# B&R Automation Studio project NewPendant_NG4_11_05_25A (part 3)

### Hardcoded.c
```c
/********************************************************************
 * COPYRIGHT -- wsi
 ********************************************************************
 * Package: Robot
 * File: Hardcoded.c
 * Author: wsi
 * Created: March 08, 2013
 *******************************************************************/
#ifndef _HARDCODED_C
#define _HARDCODED_C

#include <bur/plctypes.h>
#ifdef _DEFAULT_INCLUDES
	#include <AsDefault.h>
#endif

#include <..\GlobDef.h>
#include <..\GlobDecl.h>
#include <..\..\Lib\LCDLib.c>

//#include <string.h>

/**
char line[6][4] = {	{0xFF,0xFF,0xFF,0x00},
					{0xFF,0xFF,0xFF,0x00},
					{0xFF,0xFF,0xFF,0x00},
					{0xFF,0xFF,0xFF,0x00},
					{0xFF,0xFF,0xFF,0x00},
					{0xFF,0xFF,0xFF,0x00} };

char emptyLine[21] = { 0x20 , 0x00 };

**/

static	plcstring txt_example[32];
static	plcstring txt_hidden_example[32];

void HardCodeCFg(MASTER_typ *m);

void SetupNODES_Android(MASTER_typ *m , UDINT pNode ,UINT nodeNum );

void SetPageDict(PAGE_DICT_typ* dict , UINT indx , char* pTxt);

void SetupNODES_Android(MASTER_typ *m , UDINT pNode ,UINT nodeNum ){

int i, k , h , n;
char status;
Cfg_typ *cfg;
CurCfg_typ *curCfg;
CurCalib_typ *curCalib;
Scaled_Var_obj *var , *tempVar;

Enum_Var_obj  *enumVar;
Integer_Var_obj *intVar;

LCD_NODE_obj *node , *tempNode;
//LCD_MGR_obj *lcd;

	if(!m)
		return;

	if(!pNode)
		return;

	node = (LCD_NODE_obj*)pNode;
	cfg = (Cfg_typ*) m->pCfg;
	curCfg = (CurCfg_typ*) m->pCurCfg;
	var = (Scaled_Var_obj*) m->pScaledVar;
	curCalib = (CurCalib_typ*) m->pCalib;

	enumVar = cfg->EnumVar;

	if(!cfg || ! curCfg || !var || !curCalib)
		return;

	/************************************/

	n = 0;

	///// MENU ////////////
	/** P_MENU **/
	i = P_MENU;			h=varSTRING_HMI_0;
	SetPageDict(&cfg->PagesDict[n++] , P_MENU , "P_MENU");

	node[i].pHeadNode	= (UDINT)&node[P_MENU];
	node[i].Type = N_SCROLL   ;
	node[i].var.Type = T_STRING;
	node[i].var.Var1ID = varSTRING_curProgramName;
	strcpy(node[i++].var.Format, "Cur Program: %s");

	node[i].pHeadNode	= (UDINT)&node[P_MENU];
	node[i].Type = N_SCROLL;
	node[i].var.Type = T_STRING;
	node[i].var.Var1ID = varSTRING_NextProgramName;
	strcpy(node[i++].var.Format, "Next Program: %s");

	node[i].pHeadNode	= (UDINT)&node[P_MENU];
	node[i].Type = N_JUMP + N_EVENT;
	node[i].Event = EVNT_EDIT_PARAM_VAL;
	node[i].JumpLineID = 0;
	node[i].MinUserLevel = USER_OPERATOR;
	node[i].pJumpNode = (UDINT)&node[P_PARAM];
	strcpy(node[i++].var.Format, "Parameters Value");

	node[i].pHeadNode	= (UDINT)&node[P_MENU];
	node[i].Type = N_JUMP + N_EVENT;
	node[i].Event = EVNT_EDIT_PARAM_VAL;
	node[i].JumpLineID = 0;
	node[i].MinUserLevel = USER_OPERATOR;
	node[i].pJumpNode = (UDINT)&node[P_PARAM_BOOSTS];
	strcpy(node[i++].var.Format, "Parameters Boost");

	node[i].pHeadNode	= (UDINT)&node[P_MENU];
	node[i].Type = N_JUMP + N_EVENT;
	node[i].Event = EVNT_EDIT_PARAM_VAL;
	node[i].JumpLineID = 0;
	node[i].MinUserLevel = USER_OPERATOR;
	node[i].pJumpNode = (UDINT)&node[P_PARAM_CONTIN_WELD];
	strcpy(node[i++].var.Format, "Parameters Contin. Weld");

	node[i].pHeadNode	= (UDINT)&node[P_MENU];
	node[i].Type = N_JUMP;
	node[i].JumpLineID = 0;
	node[i].MinUserLevel = USER_OPERATOR;
	node[i].pJumpNode = (UDINT)&node[P_PAR_REVIEW];
	strcpy(node[i++].var.Format, "Timing Review");

	node[i].pHeadNode	= (UDINT)&node[P_MENU];
	node[i].Type = N_JUMP;
	node[i].JumpLineID = 0;
	node[i].MinUserLevel = USER_OPERATOR;
	node[i].pJumpNode = (UDINT)&node[P_VAR_SETUP];
	strcpy(node[i++].var.Format, "Var Unit Setup");

	node[i].pHeadNode	= (UDINT)&node[P_MENU];
	node[i].Type = N_JUMP;
	node[i].JumpLineID = 0;
	node[i].MinUserLevel = USER_OPERATOR;
	node[i].pJumpNode = (UDINT)&node[P_SPEC_OPERATION];
	strcpy(node[i++].var.Format, "Special Operation");

	node[i].pHeadNode 	= (UDINT)&node[P_MENU];
	node[i].Type = N_SCROLL + N_NO_PREFIX;
	node[i].var.Type = T_STRING;
	node[i].var.Var1ID = varSTRING_PlcVersion;
	strcpy(node[i++].var.Format, "%s");

	node[i].pHeadNode	= (UDINT)&node[P_MENU];
	node[i].Type = N_SCROLL + N_EVENT ;
	node[i].Event = EVNT_TOGGLE;
	node[i].var.Type = T_STRING;
	node[i].var.Var1ID = (h++);
	strcpy(node[i++].var.Format, "COOL PWR is: %s");

	node[i].pHeadNode	= (UDINT)&node[P_MENU];
	node[i].Type = N_SCROLL  + N_EDIT_IN_PLACE ;
	node[i].var.Type = T_STRING;
	node[i].var.Var1ID = (h++);
	strcpy(node[i++].var.Format, "COOL Sensor is: %s");

	node[i].pHeadNode	= (UDINT)&node[P_MENU];
	node[i].Type = N_SCROLL  + N_EDIT_IN_PLACE ;
	node[i].var.Type = T_STRING;
	node[i].var.Var1ID = (h++);
	strcpy(node[i++].var.Format, "GAS Sensor is: %s");

	////

	/*
	node[i].pHeadNode	= (UDINT)&node[P_MENU];
	node[i].Type = N_JUMP;
	node[i].JumpLineID = 0;
	node[i].MinUserLevel = USER_OPERATOR;
	node[i].pJumpNode = (UDINT)&node[P_SEGMENTS];
	strcpy(node[i++].var.Format, "Segments Setup");
	*/

	/** P_MODE_CALIB**/
	i = P_MODE_CALIB;			h=varSTRING_HMI_0;
	SetPageDict(&cfg->PagesDict[n++] , P_MODE_CALIB , "P_MODE_CALIB");

	node[i].pHeadNode	= (UDINT)&node[P_MODE_CALIB];
	node[i].Type = N_JUMP + N_EVENT;
	node[i].Event = EVNT_RETURN_CALIB_MODE;
	node[i].MinUserLevel = USER_OPERATOR;
	node[i].pJumpNode = (UDINT)&node[P_MENU];
	strcpy(node[i++].var.Format, "Return ");

	node[i].pHeadNode	= (UDINT)&node[P_MODE_CALIB];
	node[i].Type = N_JUMP + N_EVENT;
	node[i].Event = EVNT_GO_CALIB_MODE;
	node[i].JumpLineID = 0;
	node[i].pJumpNode = (UDINT)&node[P_MODE_TIG_PS_CALIB_PAR];
	strcpy(node[i++].var.Format, "TIG PS Calib.");

	node[i].pHeadNode	= (UDINT)&node[P_MODE_CALIB];
	node[i].Type = N_JUMP + N_EVENT;
	node[i].Event = EVNT_GO_CALIB_MODE;
	node[i].JumpLineID = 0;
	node[i].pJumpNode = (UDINT)&node[P_MODE_HW_PS_CALIB_PAR];
	strcpy(node[i++].var.Format, "HW PS Calib");

	node[i].pHeadNode	= (UDINT)&node[P_MODE_CALIB];
	node[i].Type = N_JUMP + N_EVENT;
	node[i].Event = EVNT_GO_CALIB_MODE;
	node[i].JumpLineID = 0;
	node[i].pJumpNode = (UDINT)&node[P_MODE_OSC_LIMIT_CALIB];
	strcpy(node[i++].var.Format, "OSC Limit Setup");

	node[i].pHeadNode	= (UDINT)&node[P_MODE_CALIB];
	node[i].Type = N_JUMP + N_EVENT;
	node[i].Event = EVNT_GO_CALIB_MODE;
	node[i].JumpLineID = 0;
	node[i].pJumpNode = (UDINT)&node[P_MODE_TIG_FBK_CALIB];
	strcpy(node[i++].var.Format, "ARC Volt FBK Calib");

	node[i].pHeadNode	= (UDINT)&node[P_MODE_CALIB];
	node[i].Type = N_JUMP + N_EVENT;
	node[i].Event = EVNT_GO_CALIB_MODE;
	node[i].JumpLineID = 0;
	node[i].pJumpNode = (UDINT)&node[P_MODE_TVL_CALIB_PAR];
	strcpy(node[i++].var.Format, "TVL Calib");

	node[i].pHeadNode	= (UDINT)&node[P_MODE_CALIB];
	node[i].Type = N_JUMP + N_EVENT;
	node[i].Event = EVNT_GO_CALIB_MODE;
	node[i].JumpLineID = 0;
	node[i].pJumpNode = (UDINT)&node[P_MODE_WF_CALIB_PAR];
	strcpy(node[i++].var.Format, "WFeed Calib");

	node[i].pHeadNode	= (UDINT)&node[P_MODE_CALIB];
	node[i].Type = N_JUMP + N_EVENT;
	node[i].Event = EVNT_VER_TIG_PS_CALIB;
	node[i].JumpLineID = 0;
	node[i].pJumpNode = (UDINT)&node[P_MODE_TIG_PS_CALIB_VER];
	strcpy(node[i++].var.Format, "TIG PS Test");

	node[i].pHeadNode	= (UDINT)&node[P_MODE_CALIB];
	node[i].Type = N_JUMP + N_EVENT;
	node[i].Event = EVNT_VER_HW_PS_CALIB;
	node[i].JumpLineID = 0;
	node[i].pJumpNode = (UDINT)&node[P_MODE_HW_PS_CALIB_VER];
	strcpy(node[i++].var.Format, "HW PS Test");

	node[i].pHeadNode	= (UDINT)&node[P_MODE_CALIB];
	node[i].Type = N_JUMP + N_EVENT;
	node[i].Event = EVNT_VER_TVL_CALIB;
	node[i].JumpLineID = 0;
	node[i].pJumpNode = (UDINT)&node[P_MODE_TVL_CALIB_VER];
	strcpy(node[i++].var.Format, "TVL Test");

	node[i].pHeadNode	= (UDINT)&node[P_MODE_CALIB];
	node[i].Type = N_JUMP + N_EVENT;
	node[i].Event = EVNT_VER_WF_CALIB;
	node[i].JumpLineID = 0;
	node[i].pJumpNode = (UDINT)&node[P_MODE_WF_CALIB_VER];
	strcpy(node[i++].var.Format, "WFeed Test");

	/** P_PARAM **/
	i = P_PARAM;			h=varSTRING_HMI_0;
	SetPageDict(&cfg->PagesDict[n++] , P_PARAM , "P_PARAM");

	node[i].pHeadNode	= (UDINT)&node[P_PARAM];
	node[i].Type = N_JUMP;
	node[i].JumpLineID = 0;
	node[i].pJumpNode = (UDINT)&node[P_MENU];
	strcpy(node[i++].var.Format, "Return ");

	node[i].pHeadNode	= (UDINT)&node[P_PARAM];
	node[i].Type = N_JUMP;
	node[i].JumpLineID = 0;
	node[i].pJumpNode = (UDINT)&node[P_PARAM_GAS];
	strcpy(node[i++].var.Format, "Param. GAS/COOL");

	node[i].pHeadNode	= (UDINT)&node[P_PARAM];
	node[i].Type = N_JUMP;
	node[i].JumpLineID = 0;
	node[i].pJumpNode = (UDINT)&node[P_PARAM_AVC];
	strcpy(node[i++].var.Format, "Param. AVC");

	node[i].pHeadNode	= (UDINT)&node[P_PARAM];
	node[i].Type = N_JUMP;
	node[i].JumpLineID = 0;
	node[i].pJumpNode = (UDINT)&node[P_PARAM_TIG];
	strcpy(node[i++].var.Format, "Param. TIG");

	node[i].pHeadNode	= (UDINT)&node[P_PARAM];
	node[i].Type = N_JUMP;
	node[i].JumpLineID = 0;
	node[i].pJumpNode = (UDINT)&node[P_PARAM_OSC];
	strcpy(node[i++].var.Format, "Param. OSC");

	node[i].pHeadNode	= (UDINT)&node[P_PARAM];
	node[i].Type = N_JUMP;
	node[i].JumpLineID = 0;
	node[i].pJumpNode = (UDINT)&node[P_PARAM_TVL_ROT];
	strcpy(node[i++].var.Format, "Param.TVL");

	node[i].pHeadNode	= (UDINT)&node[P_PARAM];
	node[i].Type = N_JUMP;
	node[i].JumpLineID = 0;
	node[i].pJumpNode = (UDINT)&node[P_PARAM_WF];
	strcpy(node[i++].var.Format, "Param. WF");

	node[i].pHeadNode	= (UDINT)&node[P_PARAM];
	node[i].Type = N_JUMP;
	node[i].JumpLineID = 0;
	node[i].pJumpNode = (UDINT)&node[P_PARAM_WP];
	strcpy(node[i++].var.Format, "Param. WP");

	node[i].pHeadNode	= (UDINT)&node[P_PARAM];
	node[i].Type = N_JUMP;
	node[i].JumpLineID = 0;
	node[i].pJumpNode = (UDINT)&node[P_PARAM_HW];
	strcpy(node[i++].var.Format, "Param. HW");

	node[i].pHeadNode	= (UDINT)&node[P_PARAM];
	node[i].Type = N_JUMP;
	node[i].JumpLineID = 0;
	node[i].pJumpNode = (UDINT)&node[P_PARAM_WRST];
	strcpy(node[i++].var.Format, "Param. WRIST");

	node[i].pHeadNode	= (UDINT)&node[P_PARAM];
	node[i].Type = N_JUMP;
	node[i].JumpLineID = 0;
	node[i].pJumpNode = (UDINT)&node[P_PARAM_INDX];
	strcpy(node[i++].var.Format, "Param. INDX");

	node[i].pHeadNode	= (UDINT)&node[P_PARAM];
	node[i].Type = N_EDIT;
	node[i].MinUserLevel = 5;
	node[i].var.Type = T_ENUM;
	node[i].var.Var1ID = parENUM_WeldProgramLinkMode;
	//strcpy(node[i++].var.Format, "Load Next Prg.: %s");
	strcpy(node[i++].var.Format, "%name%: %s");

	node[i].pHeadNode	= (UDINT)&node[P_PARAM];
	node[i].Type = N_EDIT;
	node[i].MinUserLevel = 5;
	node[i].var.Type = T_ENUM;
	node[i].var.Var1ID = parENUM_PathMode;
	//strcpy(node[i++].var.Format, "Swap Head: %s");
	strcpy(node[i++].var.Format, "%name%: %s");

	node[i].pHeadNode	= (UDINT)&node[P_PARAM];
	node[i].Type = N_EDIT;
	node[i].var.Type = T_SCALED;
	node[i].var.Var1ID = parGEN_WeldProgramRepeat;
	//strcpy(node[i++].var.Format, "Repeat: %s");
	strcpy(node[i++].var.Format, "%name%: %s");

	node[i].pHeadNode	= (UDINT)&node[P_PARAM];
	node[i].Type = N_SCROLL + N_EDIT_IN_PLACE;
	node[i].var.Type = T_STRING;
	node[i].var.Var1ID = (h++);
	strcpy(node[i++].var.Format, "%s");

	node[i].pHeadNode 	= (UDINT)&node[P_PARAM];
	node[i].Type = N_SCROLL + N_NO_PREFIX;
	node[i].MinUserLevel = 5;
	strcpy(node[i++].var.Format, "** SYNCH. options**");

	node[i].pHeadNode	= (UDINT)&node[P_PARAM];
	node[i].Type = N_EDIT;
	node[i].MinUserLevel = 5;
	node[i].var.Type = T_ENUM;
	node[i].var.Var1ID = parENUM_TIG_Mode;
	//strcpy(node[i++].var.Format, "TIG Mode: %s");
	strcpy(node[i++].var.Format, "%name%: %s");

	node[i].pHeadNode	= (UDINT)&node[P_PARAM];
	node[i].Type = N_EDIT;
	node[i].MinUserLevel = 5;
	node[i].var.Type = T_ENUM;
	node[i].var.Var1ID = parENUM_AVC_Mode;
	//strcpy(node[i++].var.Format, "AVC Mode: %s");
	strcpy(node[i++].var.Format, "%name%: %s");

	node[i].pHeadNode	= (UDINT)&node[P_PARAM];
	node[i].Type = N_EDIT;
	node[i].MinUserLevel = 5;
	node[i].var.Type = T_ENUM;
	node[i].var.Var1ID = parENUM_TVL_SYN_MODE;
	//strcpy(node[i++].var.Format, "TVL Synch. Mode: %s");
	strcpy(node[i++].var.Format, "%name%: %s");

	node[i].pHeadNode	= (UDINT)&node[P_PARAM];
	node[i].Type = N_EDIT;
	node[i].MinUserLevel = 5;
	node[i].var.Type = T_ENUM;
	node[i].var.Var1ID = parENUM_WF_SYN_MODE;
	//strcpy(node[i++].var.Format, "WF Synch. Mode: %s");
	strcpy(node[i++].var.Format, "%name%: %s");

	node[i].pHeadNode	= (UDINT)&node[P_PARAM];
	node[i].Type = N_EDIT;
	node[i].MinUserLevel = 5;
	node[i].var.Type = T_ENUM;
	node[i].var.Var1ID = parENUM_WP_SYN_MODE;
	//strcpy(node[i++].var.Format, "WP Synch. Mode: %s");
	strcpy(node[i++].var.Format, "%name%: %s");

	i = P_PARAM_APPL;			h=varSTRING_HMI_0;
	SetPageDict(&cfg->PagesDict[n++] , P_PARAM_APPL , "P_PARAM_APPL");

	node[i].pHeadNode	= (UDINT)&node[P_PARAM_APPL];
	node[i].Type = N_EDIT;
	node[i].MinUserLevel = 5;
	node[i].var.Type = T_SCALED;
	node[i].var.Var1ID = parTVL_RunDist;
	//strcpy(node[i++].var.Format, "RUN Dist: %s");
	strcpy(node[i++].var.Format, "%name%: %s");

	node[i].pHeadNode	= (UDINT)&node[P_PARAM_APPL];
	node[i].Type = N_SCROLL + N_EDIT_IN_PLACE;
	node[i].MinUserLevel = 5;
	node[i].var.Type = T_STRING;
	node[i].var.Var1ID = (h++);
	strcpy(node[i++].var.Format, "%s"); // Zone editor

	node[i].pHeadNode	= (UDINT)&node[P_PARAM_APPL];
	node[i].Type = N_SCROLL + N_EDIT_IN_PLACE;
	node[i].MinUserLevel = 5;
	node[i].var.Type = T_STRING;
	node[i].var.Var1ID = (h++);
	strcpy(node[i++].var.Format, "%s"); // Track Dia

	node[i].pHeadNode	= (UDINT)&node[P_PARAM_APPL];
	node[i].Type = N_EDIT;
	node[i].var.Type = T_SCALED;
	node[i].var.Var1ID = parTVL_TrackDia;
	//strcpy(node[i++].var.Format, "Tungsten Track Dia: %s");
	strcpy(node[i++].var.Format, "%name%: %s");

	node[i].pHeadNode	= (UDINT)&node[P_PARAM_APPL];
	node[i].Type = N_EDIT;
	node[i].MinUserLevel = 5;
	node[i].var.Type = T_ENUM;
	node[i].var.Var1ID = parENUM_WeldProgramLinkMode;
	//strcpy(node[i++].var.Format, "Load Next Prg.: %s");
	strcpy(node[i++].var.Format, "%name%: %s");

	node[i].pHeadNode	= (UDINT)&node[P_PARAM_APPL];
	node[i].Type = N_EDIT;
	node[i].MinUserLevel = 5;
	node[i].var.Type = T_ENUM;
	node[i].var.Var1ID = parENUM_PathMode;
	//strcpy(node[i++].var.Format, "Swap Head: %s");
	strcpy(node[i++].var.Format, "%name%: %s");

	node[i].pHeadNode	= (UDINT)&node[P_PARAM_APPL];
	node[i].Type = N_EDIT;
	node[i].var.Type = T_SCALED;
	node[i].var.Var1ID = parGEN_WeldProgramRepeat;
	//strcpy(node[i++].var.Format, "Repeat: %s");
	strcpy(node[i++].var.Format, "%name%: %s");

	node[i].pHeadNode	= (UDINT)&node[P_PARAM_APPL];
	node[i].Type = N_SCROLL + N_EDIT_IN_PLACE;
	node[i].MinUserLevel = 5;
	node[i].var.Type = T_STRING;
	node[i].var.Var1ID = (h++);
	strcpy(node[i++].var.Format, "%s"); // Weld Report ON / OFF

	node[i].pHeadNode	= (UDINT)&node[P_PARAM_APPL];
	node[i].Type = N_SCROLL + N_EDIT_IN_PLACE;
	node[i].MinUserLevel = 5;
	node[i].var.Type = T_STRING;
	node[i].var.Var1ID = (h++);
	strcpy(node[i++].var.Format, "%s"); // TVL Reverse RampDown ON / OFF

	/*
	node[i].pHeadNode	= (UDINT)&node[P_PARAM_APPL];
	node[i].Type = N_SCROLL + N_EVENT;
	node[i].Event = EVNT_OK;
	node[i].MinUserLevel = 5;
	node[i].var.Type = T_STRING;
	node[i].var.Var1ID = (h++);
	strcpy(node[i++].var.Format, "%s"); // Set Tilt Zero
	*/

	/** P_PARAM_WRST **/
	i = P_PARAM_WRST;			h=varSTRING_HMI_0;
	SetPageDict(&cfg->PagesDict[n++] , P_PARAM_WRST , "P_PARAM_WRST");

	node[i].pHeadNode	= (UDINT)&node[P_PARAM_WRST];
	node[i].Type = N_JUMP;
	node[i].JumpLineID = 0;
	node[i].pJumpNode = (UDINT)&node[P_PARAM];
	strcpy(node[i++].var.Format, "Return ");

	node[i].pHeadNode 	= (UDINT)&node[P_PARAM_WRST];
	node[i].Type = N_EDIT;
	node[i].MinUserLevel = 5;
	node[i].var.Type = T_SCALED;
	node[i].var.Var1ID = parWRST_JogSpeedDirCntrl;
	strcpy(node[i++].var.Format, "%name%: %s");

	node[i].pHeadNode 	= (UDINT)&node[P_PARAM_WRST];
	node[i].Type = N_EDIT;
	node[i].MinUserLevel = 5;
	node[i].var.Type = T_SCALED;
	node[i].var.Var1ID = parGEN_RadSpeed_Boost;
	strcpy(node[i++].var.Format, "%name%: %s");

	node[i].pHeadNode 	= (UDINT)&node[P_PARAM_WRST];
	node[i].Type = N_EDIT;
	node[i].MinUserLevel = 5;
	node[i].var.Type = T_SCALED;
	node[i].var.Var1ID = parTVL_POS_PREDICT;
	strcpy(node[i++].var.Format, "%name%: %s");

	node[i].pHeadNode	= (UDINT)&node[P_PARAM_WRST];
	node[i].Type = N_SCROLL;
	node[i].var.Type = T_STRING;
	node[i].var.Var1ID = (h++);
	strcpy(node[i++].var.Format, "%s");

	node[i].pHeadNode	= (UDINT)&node[P_PARAM_WRST];
	node[i].Type = N_SCROLL +  N_EVENT ;
	node[i].Event = EVNT_OK;
	node[i].var.Type = T_STRING;
	node[i].var.Var1ID = (h++);
	strcpy(node[i++].var.Format, "%s");

	/** P_PARAM_OSC **/
	i = P_PARAM_OSC;			h=varSTRING_HMI_0;
	SetPageDict(&cfg->PagesDict[n++] , P_PARAM_OSC , "P_PARAM_OSC");

	node[i].pHeadNode	= (UDINT)&node[P_PARAM_OSC];
	node[i].Type = N_JUMP;
	node[i].JumpLineID = 0;
	node[i].pJumpNode = (UDINT)&node[P_PARAM];
	strcpy(node[i++].var.Format, "Return ");

	node[i].pHeadNode 	= (UDINT)&node[P_PARAM_OSC];
	node[i].Type = N_EDIT;
	node[i].MinUserLevel = 5;
	node[i].var.Type = T_SCALED;
	node[i].var.Var1ID = parOSC_Amplit;
	//strcpy(node[i++].var.Format, "OSC WIDTH %s");
	strcpy(node[i++].var.Format, "%name%: %s");

	node[i].pHeadNode 	= (UDINT)&node[P_PARAM_OSC];
	node[i].Type = N_EDIT;
	node[i].MinUserLevel = 5;
	node[i].var.Type = T_SCALED;
	node[i].var.Var1ID = parOSC_Excur;
	//strcpy(node[i++].var.Format, "Excurs Tm.: %s");
	strcpy(node[i++].var.Format, "%name%: %s");

	node[i].pHeadNode 	= (UDINT)&node[P_PARAM_OSC];
	node[i].Type = N_EDIT;
	node[i].MinUserLevel = 5;
	node[i].var.Type = T_SCALED;
	node[i].var.Var1ID = parOSC_Dwell_In;
	//strcpy(node[i++].var.Format, "Dwell In: %s");
	strcpy(node[i++].var.Format, "%name%: %s");

	node[i].pHeadNode 	= (UDINT)&node[P_PARAM_OSC];
	node[i].Type = N_EDIT;
	node[i].MinUserLevel = 5;
	node[i].var.Type = T_SCALED;
	node[i].var.Var1ID = parOSC_Dwell_Out;
	//strcpy(node[i++].var.Format, "Dwell Out: %s");
	strcpy(node[i++].var.Format, "%name%: %s");

	node[i].pHeadNode 	= (UDINT)&node[P_PARAM_OSC];
	node[i].Type = N_SCROLL + N_NO_PREFIX;
	node[i].MinUserLevel = 5;
	strcpy(node[i++].var.Format, "******* MSC. *******");

	node[i].pHeadNode 	= (UDINT)&node[P_PARAM_OSC];
	node[i].Type = N_EDIT;
	node[i].MinUserLevel = 5;
	node[i].var.Type = T_SCALED;
	node[i].var.Var1ID = parOSC_InitAmplit;
	//strcpy(node[i++].var.Format, "OSC INI W %s");
	strcpy(node[i++].var.Format, "%name%: %s");

	node[i].pHeadNode 	= (UDINT)&node[P_PARAM_OSC];
	node[i].Type = N_EDIT;
	node[i].MinUserLevel = 5;
	node[i].var.Type = T_SCALED;
	node[i].var.Var1ID = parOSC_FinalAmplit;
	//strcpy(node[i++].var.Format, "OSC FIN W %s");
	strcpy(node[i++].var.Format, "%name%: %s");

	node[i].pHeadNode 	= (UDINT)&node[P_PARAM_OSC];
	node[i].Type = N_EDIT;
	node[i].MinUserLevel = 5;
	node[i].var.Type = T_ENUM;
	node[i].var.Var1ID = parENUM_OSC_Mode;
	strcpy(node[i++].var.Format, "%name%: %s");

	node[i].pHeadNode 	= (UDINT)&node[P_PARAM_OSC];
	node[i].Type = N_EDIT;
	node[i].MinUserLevel = 5;
	node[i].var.Type = T_ENUM;
	node[i].var.Var1ID = parENUM_OSC_Synch;
	strcpy(node[i++].var.Format, "%name%: %s");

	node[i].pHeadNode 	= (UDINT)&node[P_PARAM_OSC];
	node[i].Type = N_EDIT;
	node[i].MinUserLevel = 5;
	node[i].var.Type = T_SCALED;
	node[i].var.Var1ID = parOSC_Indx;
	strcpy(node[i++].var.Format, "%name%: %s");

	node[i].pHeadNode 	= (UDINT)&node[P_PARAM_OSC];
	node[i].Type = N_EDIT;
	node[i].MinUserLevel = 5;
	node[i].var.Type = T_SCALED;
	node[i].var.Var1ID = parOSC_Period;
	strcpy(node[i++].var.Format, "%name%: %s");

	node[i].pHeadNode 	= (UDINT)&node[P_PARAM_OSC];
	node[i].Type = N_EDIT;
	node[i].MinUserLevel = 5;
	node[i].var.Type = T_SCALED;
	node[i].var.Var1ID = parOSC_Indx_Vel;
	strcpy(node[i++].var.Format, "%name%: %s");

	node[i].pHeadNode 	= (UDINT)&node[P_PARAM_OSC];
	node[i].Type = N_EDIT;
	node[i].MinUserLevel = 5;
	node[i].var.Type = T_SCALED;
	node[i].var.Var1ID = parOSC_RampUpdate;
	//strcpy(node[i++].var.Format, "RampUpd.: %s");
	strcpy(node[i++].var.Format, "%name%: %s");

	node[i].pHeadNode	= (UDINT)&node[P_PARAM_OSC];
	node[i].Type = N_EDIT;
	node[i].MinUserLevel = 5;
	node[i].var.Type = T_SCALED;
	node[i].var.Var1ID = parOSC_JogSpeed;
	//strcpy(node[i++].var.Format, "Steer Speed: %s");
	strcpy(node[i++].var.Format, "%name%: %s");

	node[i].pHeadNode	= (UDINT)&node[P_PARAM_OSC];
	node[i].Type = N_EDIT;
	node[i].MinUserLevel = 5;
	node[i].var.Type = T_SCALED;
	node[i].var.Var1ID = parOSC_JogSpeedDirCntrl;
	//strcpy(node[i++].var.Format, "Jog Cntrl: %s");
	strcpy(node[i++].var.Format, "%name%: %s");

	node[i].pHeadNode 	= (UDINT)&node[P_PARAM_OSC];
	node[i].Type = N_EDIT;
	node[i].MinUserLevel = 5;
	node[i].var.Type = T_ENUM;
	node[i].var.Var1ID = parENUM_OSC_CAM;
	//strcpy(node[i++].var.Format, "Cam.: %s");
	strcpy(node[i++].var.Format, "%name%: %s");

	node[i].pHeadNode	= (UDINT)&node[P_PARAM_OSC];
	node[i].Type = N_EDIT;
	node[i].MinUserLevel = 5;
	node[i].var.Type = T_SCALED;
	node[i].var.Var1ID = parOSC_MaxTvlVel;
	//strcpy(node[i++].var.Format, "Max OSC Vel: %s");
	strcpy(node[i++].var.Format, "%name%: %s");

	node[i].pHeadNode 	= (UDINT)&node[P_PARAM_OSC];
	node[i].Type = N_SCROLL + N_NO_PREFIX;
	node[i].MinUserLevel = 5;
	strcpy(node[i++].var.Format, "**** CALCULATED ****");

	node[i].pHeadNode	= (UDINT)&node[P_PARAM_OSC];
	node[i].Type = N_EDIT;
	node[i].MinUserLevel = 5;
	node[i].var.Type = T_SCALED;
	node[i].var.Var1ID = parOSC_StartDly;
	//strcpy(node[i++].var.Format, "OSC DLY %s");
	strcpy(node[i++].var.Format, "%name%: %s");

	node[i].pHeadNode 	= (UDINT)&node[P_PARAM_OSC];
	node[i].Type = N_EDIT;
	node[i].MinUserLevel = 5;
	node[i].var.Type = T_SCALED;
	node[i].var.Var1ID = parOSC_RampUp;
	//strcpy(node[i++].var.Format, "O UPSCLOPE %s");
	strcpy(node[i++].var.Format, "%name%: %s");

	node[i].pHeadNode 	= (UDINT)&node[P_PARAM_OSC];
	node[i].Type = N_EDIT;
	node[i].MinUserLevel = 5;
	node[i].var.Type = T_SCALED;
	node[i].var.Var1ID = parOSC_StopDly;
	//strcpy(node[i++].var.Format, "O DS DLY %s");
	strcpy(node[i++].var.Format, "%name%: %s");

	node[i].pHeadNode 	= (UDINT)&node[P_PARAM_OSC];
	node[i].Type = N_EDIT;
	node[i].MinUserLevel = 5;
	node[i].var.Type = T_SCALED;
	node[i].var.Var1ID = parOSC_RampDwn;
	//strcpy(node[i++].var.Format, "O DWNSLOP %s");
	strcpy(node[i++].var.Format, "%name%: %s");

	/** P_PARAM_TVL_ROT **/
	i = P_PARAM_TVL_ROT;			h=varSTRING_HMI_0;
	SetPageDict(&cfg->PagesDict[n++] , P_PARAM_TVL_ROT , "P_PARAM_TVL_ROT");

	node[i].pHeadNode	= (UDINT)&node[P_PARAM_TVL_ROT];
	node[i].Type = N_JUMP;
	node[i].JumpLineID = 0;
	node[i].pJumpNode = (UDINT)&node[P_PARAM];
	strcpy(node[i++].var.Format, "Return ");

	node[i].pHeadNode 	= (UDINT)&node[P_PARAM_TVL_ROT];
	node[i].Type = N_EDIT;
	node[i].MinUserLevel = 5;
	node[i].var.Type = T_SCALED;
	node[i].var.Var1ID = parTVL_VelSP;
	node[i].var.Type = T_SCALED;
	//strcpy(node[i++].var.Format, "T PRI SP %s");
	strcpy(node[i++].var.Format, "%name%: %s");

	node[i].pHeadNode 	= (UDINT)&node[P_PARAM_TVL_ROT];
	node[i].Type = N_EDIT;
	node[i].MinUserLevel = 5;
	node[i].var.Type = T_SCALED;
	node[i].var.Var1ID = parTVL_VelInSP;
	node[i].var.Type = T_SCALED;
	//strcpy(node[i++].var.Format, "T PRI IN SP %s");
	strcpy(node[i++].var.Format, "%name%: %s");

	node[i].pHeadNode 	= (UDINT)&node[P_PARAM_TVL_ROT];
	node[i].Type = N_EDIT;
	node[i].MinUserLevel = 5;
	node[i].var.Type = T_SCALED;
	node[i].var.Var1ID = parTVL_VelOutSP;
	node[i].var.Type = T_SCALED;
	//strcpy(node[i++].var.Format, "T PRI OUT SP %s");
	strcpy(node[i++].var.Format, "%name%: %s");

	node[i].pHeadNode 	= (UDINT)&node[P_PARAM_TVL_ROT];
	node[i].Type = N_EDIT;
	node[i].MinUserLevel = 5;
	node[i].var.Type = T_SCALED;
	node[i].var.Var1ID = parTVL_VelBackSP;
	node[i].var.Type = T_SCALED;
	//strcpy(node[i++].var.Format, "T BCKG SP %s");
	strcpy(node[i++].var.Format, "%name%: %s");

	node[i].pHeadNode	= (UDINT)&node[P_PARAM_TVL_ROT];
	node[i].Type = N_EDIT;
	node[i].MinUserLevel = 5;
	node[i].var.Type = T_SCALED;
	node[i].var.Var1ID = parTVL_OverlapDist;
	//strcpy(node[i++].var.Format, "OVERLAP DIST: %s");
	strcpy(node[i++].var.Format, "%name%: %s");

	node[i].pHeadNode 	= (UDINT)&node[P_PARAM_TVL_ROT];
	node[i].Type = N_SCROLL + N_NO_PREFIX;
	node[i].MinUserLevel = 5;
	strcpy(node[i++].var.Format, "******* MSC. *******");

	node[i].pHeadNode 	= (UDINT)&node[P_PARAM_TVL_ROT];
	node[i].Type = N_EDIT;
	node[i].MinUserLevel = 5;
	node[i].var.Type = T_SCALED;
	node[i].var.Var1ID = parTVL_InitVel;
	node[i].var.Type = T_SCALED;
	//strcpy(node[i++].var.Format, "T INI SP %s");
	strcpy(node[i++].var.Format, "%name%: %s");

	node[i].pHeadNode 	= (UDINT)&node[P_PARAM_TVL_ROT];
	node[i].Type = N_EDIT;
	node[i].MinUserLevel = 5;
	node[i].var.Type = T_SCALED;
	node[i].var.Var1ID = parTVL_FinalVel;
	node[i].var.Type = T_SCALED;
	//strcpy(node[i++].var.Format, "T FIN SP %s");
	strcpy(node[i++].var.Format, "%name%: %s");

	node[i].pHeadNode 	= (UDINT)&node[P_PARAM_TVL_ROT];
	node[i].Type = N_EDIT;
	node[i].MinUserLevel = 5;
	node[i].var.Type = T_SCALED;
	node[i].var.Var1ID = parTVL_RampUpdate;
	//strcpy(node[i++].var.Format, "RampUpd.: %s");
	strcpy(node[i++].var.Format, "%name%: %s");

	node[i].pHeadNode	= (UDINT)&node[P_PARAM_TVL_ROT];
	node[i].Type = N_EDIT;
	node[i].MinUserLevel = 5;
	node[i].var.Type = T_SCALED;
	node[i].var.Var1ID = parTVL_JogSpeedDirCntrl;
	//strcpy(node[i++].var.Format, "Jog Cntrl: %s");
	strcpy(node[i++].var.Format, "%name%: %s");

	node[i].pHeadNode	= (UDINT)&node[P_PARAM_TVL_ROT];
	node[i].Type = N_EDIT;
	node[i].MinUserLevel = 5;
	node[i].var.Type = T_SCALED;
	node[i].var.Var1ID = parTVL_RewrapVel;
	//strcpy(node[i++].var.Format, "REWRP SP %s");
	strcpy(node[i++].var.Format, "%name%: %s");

	node[i].pHeadNode	= (UDINT)&node[P_PARAM_TVL_ROT];
	node[i].Type = N_EDIT;
	node[i].MinUserLevel = 5;
	node[i].var.Type = T_ENUM;
	node[i].var.Var1ID = parENUM_TVL_MODE;
	//strcpy(node[i++].var.Format, "TVL Mode: %s");
	strcpy(node[i++].var.Format, "%name%: %s");

	node[i].pHeadNode	= (UDINT)&node[P_PARAM_TVL_ROT];
	node[i].Type = N_EDIT;
	node[i].MinUserLevel = 5;
	node[i].var.Type = T_SCALED;
	node[i].var.Var1ID = parTVL_Jog2Stop;
	//strcpy(node[i++].var.Format, "Jog2Stop: %s");
	strcpy(node[i++].var.Format, "%name%: %s");

	node[i].pHeadNode	= (UDINT)&node[P_PARAM_TVL_ROT];
	node[i].Type = N_EDIT;
	node[i].MinUserLevel = 5;
	node[i].var.Type = T_SCALED;
	node[i].var.Var1ID = parTVL_SpeedTolerane;
	//strcpy(node[i++].var.Format, "Vel Toler: %s");
	strcpy(node[i++].var.Format, "%name%: %s");

	node[i].pHeadNode	= (UDINT)&node[P_PARAM_TVL_ROT];
	node[i].Type = N_EDIT;
	node[i].var.Type = T_SCALED;
	node[i].var.Var1ID = parTVL_CalibVel1;
	//strcpy(node[i++].var.Format, "Cal Vel1: %s");
	strcpy(node[i++].var.Format, "%name%: %s");

	node[i].pHeadNode	= (UDINT)&node[P_PARAM_TVL_ROT];
	node[i].Type = N_EDIT;
	node[i].var.Type = T_SCALED;
	node[i].var.Var1ID = parTVL_CalibVel2;
	//strcpy(node[i++].var.Format, "Cal Vel2: %s");
	strcpy(node[i++].var.Format, "%name%: %s");

	node[i].pHeadNode	= (UDINT)&node[P_PARAM_TVL_ROT];
	node[i].Type = N_EDIT;
	node[i].var.Type = T_SCALED;
	node[i].var.Var1ID = parTVL_TrackDia;
	//strcpy(node[i++].var.Format, "Tungsten Track Dia: %s");
	strcpy(node[i++].var.Format, "%name%: %s");

	node[i].pHeadNode	= (UDINT)&node[P_PARAM_TVL_ROT];
	node[i].Type = N_SCROLL + N_NO_PREFIX;
	node[i].MinUserLevel = 5;
	strcpy(node[i++].var.Format, "**** CALCULATED ****");

	node[i].pHeadNode 	= (UDINT)&node[P_PARAM_TVL_ROT];
	node[i].Type = N_EDIT;
	node[i].MinUserLevel = 5;
	node[i].var.Type = T_SCALED;
	node[i].var.Var1ID = parTVL_StartDly;
	//strcpy(node[i++].var.Format, "TVL DLY %s");
	strcpy(node[i++].var.Format, "%name%: %s");

	node[i].pHeadNode 	= (UDINT)&node[P_PARAM_TVL_ROT];
	node[i].Type = N_EDIT;
	node[i].MinUserLevel = 5;
	node[i].var.Type = T_SCALED;
	node[i].var.Var1ID = parTVL_RampUp;
	//strcpy(node[i++].var.Format, "T_UPSLOPE %s");
	strcpy(node[i++].var.Format, "%name%: %s");

	node[i].pHeadNode 	= (UDINT)&node[P_PARAM_TVL_ROT];
	node[i].Type = N_EDIT;
	node[i].MinUserLevel = 5;
	node[i].var.Type = T_SCALED;
	node[i].var.Var1ID = parTVL_StopDly;
	//strcpy(node[i++].var.Format, "T DS DLY %s");
	strcpy(node[i++].var.Format, "%name%: %s");

	node[i].pHeadNode 	= (UDINT)&node[P_PARAM_TVL_ROT];
	node[i].Type = N_EDIT;
	node[i].MinUserLevel = 5;
	node[i].var.Type = T_SCALED;
	node[i].var.Var1ID = parTVL_RampDwn;
	//strcpy(node[i++].var.Format, "T DWNSLOP %s");
	strcpy(node[i++].var.Format, "%name%: %s");

	node[i].pHeadNode	= (UDINT)&node[P_PARAM_TVL_ROT];
	node[i].Type = N_EDIT;
	node[i].MinUserLevel = 5;
	node[i].var.Type = T_SCALED;
	node[i].var.Var1ID = parTVL_RewrapDly;
	//strcpy(node[i++].var.Format, "REWRP DLY %s");
	strcpy(node[i++].var.Format, "%name%: %s");

	node[i].pHeadNode	= (UDINT)&node[P_PARAM_TVL_ROT];
	node[i].Type = N_EDIT;
	node[i].MinUserLevel = 5;
	node[i].var.Type = T_SCALED;
	node[i].var.Var1ID = parTVL_RunDist;
	//strcpy(node[i++].var.Format, "RUN Dist: %s");
	strcpy(node[i++].var.Format, "%name%: %s");

	node[i].pHeadNode	= (UDINT)&node[P_PARAM_TVL_ROT];
	node[i].Type = N_EDIT;
	node[i].MinUserLevel = 5;
	node[i].var.Type = T_SCALED;
	node[i].var.Var1ID = parTVL_BalanceDist;
	//strcpy(node[i++].var.Format, "Balance Dist: %s");
	strcpy(node[i++].var.Format, "%name%: %s");

	node[i].pHeadNode	= (UDINT)&node[P_PARAM_TVL_ROT];
	node[i].Type = N_EDIT;
	node[i].MinUserLevel = 5;
	node[i].var.Type = T_SCALED;
	node[i].var.Var1ID = parTVL_ZigZagDist;
	//strcpy(node[i++].var.Format, "ZigZag Dist: %s");
	strcpy(node[i++].var.Format, "%name%: %s");

	/** P_PARAM_WP **/
	i = P_PARAM_WP;			h=varSTRING_HMI_0;
	SetPageDict(&cfg->PagesDict[n++] , P_PARAM_WP , "P_PARAM_WP");

	node[i].pHeadNode	= (UDINT)&node[P_PARAM_WP];
	node[i].Type = N_JUMP;
	node[i].JumpLineID = 0;
	node[i].pJumpNode = (UDINT)&node[P_PARAM];
	strcpy(node[i++].var.Format, "Return ");

	node[i].pHeadNode	= (UDINT)&node[P_PARAM_WP];
	node[i].Type = N_EDIT;
	node[i].MinUserLevel = 5;
	node[i].var.Type = T_SCALED;
	node[i].var.Var1ID = parWP_SpeedSP;
	//strcpy(node[i++].var.Format, "WP FRG SP %s");
	strcpy(node[i++].var.Format, "%name% %s");

	node[i].pHeadNode	= (UDINT)&node[P_PARAM_WP];
	node[i].Type = N_EDIT;
	node[i].MinUserLevel = 5;
	node[i].var.Type = T_SCALED;
	node[i].var.Var1ID = parWP_SpeedInSP;
	//strcpy(node[i++].var.Format, "WP FRG IN SP %s");
	strcpy(node[i++].var.Format, "%name% %s");

	node[i].pHeadNode	= (UDINT)&node[P_PARAM_WP];
	node[i].Type = N_EDIT;
	node[i].MinUserLevel = 5;
	node[i].var.Type = T_SCALED;
	node[i].var.Var1ID = parWP_SpeedOutSP;
	//strcpy(node[i++].var.Format, "WP FRG OUT SP %s");
	strcpy(node[i++].var.Format, "%name%: %s");

	node[i].pHeadNode	= (UDINT)&node[P_PARAM_WP];
	node[i].Type = N_EDIT;
	node[i].MinUserLevel = 5;
	node[i].var.Type = T_SCALED;
	node[i].var.Var1ID = parWP_BkgSpeedSP;
	//strcpy(node[i++].var.Format, "WP BKG SP %s");
	strcpy(node[i++].var.Format, "%name%: %s");

	node[i].pHeadNode 	= (UDINT)&node[P_PARAM_WP];
	node[i].Type = N_SCROLL;
	node[i].MinUserLevel = 5;
	strcpy(node[i++].var.Format, "******* MSC. *******");

	node[i].pHeadNode	= (UDINT)&node[P_PARAM_WP];
	node[i].Type = N_EDIT;
	node[i].MinUserLevel = 5;
	node[i].var.Type = T_SCALED;
	node[i].var.Var1ID = parWP_SpeedInit;
	//strcpy(node[i++].var.Format, "WP INI SP %s");
	strcpy(node[i++].var.Format, "%name% %s");

	node[i].pHeadNode	= (UDINT)&node[P_PARAM_WP];
	node[i].Type = N_EDIT;
	node[i].MinUserLevel = 5;
	node[i].var.Type = T_SCALED;
	node[i].var.Var1ID = parWP_SpeedFinal;
	//strcpy(node[i++].var.Format, "WP FIN SP %s");
	strcpy(node[i++].var.Format, "%name%: %s");

	node[i].pHeadNode	= (UDINT)&node[P_PARAM_WP];
	node[i].Type = N_EDIT;
	node[i].MinUserLevel = 5;
	node[i].var.Type = T_SCALED;
	node[i].var.Var1ID = parWP_RampUpdate;
	//strcpy(node[i++].var.Format, "RampUpdate: %s");
	strcpy(node[i++].var.Format, "%name%: %s");

	/*
	node[i].pHeadNode	= (UDINT)&node[P_PARAM_WP];
	node[i].Type = N_EDIT;
	node[i].MinUserLevel = 5;
	node[i].var.Type = T_SCALED;
	node[i].var.Var1ID = parWP_Boost1SP;
	//strcpy(node[i++].var.Format, "Boost1: %s");
	strcpy(node[i++].var.Format, "%name% %s");

	node[i].pHeadNode	= (UDINT)&node[P_PARAM_WP];
	node[i].Type = N_EDIT;
	node[i].MinUserLevel = 5;
	node[i].var.Type = T_SCALED;
	node[i].var.Var1ID = parWP_Boost2SP;
	//strcpy(node[i++].var.Format, "Boost2: %s");
	strcpy(node[i++].var.Format, "%name% %s");
	*/

	node[i].pHeadNode	= (UDINT)&node[P_PARAM_WP];
	node[i].Type = N_EDIT;
	node[i].MinUserLevel = 5;
	node[i].var.Type = T_SCALED;
	node[i].var.Var1ID = parWP_JogSpeed;
	//strcpy(node[i++].var.Format, "Jog Vel.: %s");
	strcpy(node[i++].var.Format, "%name%: %s");

	node[i].pHeadNode	= (UDINT)&node[P_PARAM_WP];
	node[i].Type = N_EDIT;
	node[i].MinUserLevel = 5;
	node[i].var.Type = T_SCALED;
	node[i].var.Var1ID = parWP_JogSpeedDirCntrl;
	//strcpy(node[i++].var.Format, "Jog Cntrl: %s");
	strcpy(node[i++].var.Format, "%name%: %s");

	node[i].pHeadNode	= (UDINT)&node[P_PARAM_WP];
	node[i].Type = N_EDIT;
	node[i].MinUserLevel = 5;
	node[i].var.Type = T_ENUM;
	node[i].var.Var1ID = parENUM_WF_WP_Relation;
	//strcpy(node[i++].var.Format, "WP Auto Calc.: %s");
	strcpy(node[i++].var.Format, "%name% %s");

	node[i].pHeadNode	= (UDINT)&node[P_PARAM_WP];
	node[i].Type = N_SCROLL + N_NO_PREFIX;
	node[i].MinUserLevel = 5;
	strcpy(node[i++].var.Format, "**** CALCULATED ****");

	node[i].pHeadNode	= (UDINT)&node[P_PARAM_WP];
	node[i].Type = N_EDIT;
	node[i].MinUserLevel = 5;
	node[i].var.Type = T_SCALED;
	node[i].var.Var1ID = parWP_StartDly;
	//strcpy(node[i++].var.Format, "WP DLY %s");
	strcpy(node[i++].var.Format, "%name%: %s");

	node[i].pHeadNode	= (UDINT)&node[P_PARAM_WP];
	node[i].Type = N_EDIT;
	node[i].MinUserLevel = 5;
	node[i].var.Type = T_SCALED;
	node[i].var.Var1ID = parWP_RampUp;
	//strcpy(node[i++].var.Format, "WP UPSLOP %s");
	strcpy(node[i++].var.Format, "%name%: %s");

	node[i].pHeadNode	= (UDINT)&node[P_PARAM_WP];
	node[i].Type = N_EDIT;
	node[i].MinUserLevel = 5;
	node[i].var.Type = T_SCALED;
	node[i].var.Var1ID = parWP_StopDly;
	//strcpy(node[i++].var.Format, "WP DS DLY %s");
	strcpy(node[i++].var.Format, "%name%: %s");

	node[i].pHeadNode	= (UDINT)&node[P_PARAM_WP];
	node[i].Type = N_EDIT;
	node[i].MinUserLevel = 5;
	node[i].var.Type = T_SCALED;
	node[i].var.Var1ID = parWP_RampDwn;
	//strcpy(node[i++].var.Format, "WP DWNSLP %s");
	strcpy(node[i++].var.Format, "%name%: %s");

	/** P_PARAM_WF **/
	i = P_PARAM_WF;			h=varSTRING_HMI_0;
	SetPageDict(&cfg->PagesDict[n++] , P_PARAM_WF , "P_PARAM_WF");

	node[i].pHeadNode	= (UDINT)&node[P_PARAM_WF];
	node[i].Type = N_JUMP;
	node[i].JumpLineID = 0;
	node[i].pJumpNode = (UDINT)&node[P_PARAM];
	strcpy(node[i++].var.Format, "Return ");

	node[i].pHeadNode	= (UDINT)&node[P_PARAM_WF];
	node[i].Type = N_EDIT;
	node[i].MinUserLevel = 5;
	node[i].var.Type = T_SCALED;
	node[i].var.Var1ID = parWF_SpeedSP;
	//strcpy(node[i++].var.Format, "WF FRG SP %s");
	strcpy(node[i++].var.Format, "%name%: %s");

	node[i].pHeadNode	= (UDINT)&node[P_PARAM_WF];
	node[i].Type = N_EDIT;
	node[i].MinUserLevel = 5;
	node[i].var.Type = T_SCALED;
	node[i].var.Var1ID = parWF_SpeedInSP;
	//strcpy(node[i++].var.Format, "WF FRG IN SP %s");
	strcpy(node[i++].var.Format, "%name%: %s");

	node[i].pHeadNode	= (UDINT)&node[P_PARAM_WF];
	node[i].Type = N_EDIT;
	node[i].MinUserLevel = 5;
	node[i].var.Type = T_SCALED;
	node[i].var.Var1ID = parWF_SpeedOutSP;
	//strcpy(node[i++].var.Format, "WF FRG OUT SP %s");
	strcpy(node[i++].var.Format, "%name%: %s");

	node[i].pHeadNode	= (UDINT)&node[P_PARAM_WF];
	node[i].Type = N_EDIT;
	node[i].MinUserLevel = 5;
	node[i].var.Type = T_SCALED;
	node[i].var.Var1ID = parWF_BkgSpeedSP;
	//strcpy(node[i++].var.Format, "WF BKG SP %s");
	strcpy(node[i++].var.Format, "%name%: %s");

	node[i].pHeadNode 	= (UDINT)&node[P_PARAM_WF];
	node[i].Type = N_SCROLL + N_NO_PREFIX;
	node[i].MinUserLevel = 5;
	strcpy(node[i++].var.Format, "******* MSC. *******");

	node[i].pHeadNode	= (UDINT)&node[P_PARAM_WF];
	node[i].Type = N_EDIT;
	node[i].MinUserLevel = 5;
	node[i].var.Type = T_SCALED;
	node[i].var.Var1ID = parWF_SpeedInit;
	//strcpy(node[i++].var.Format, "WF INI SP %s");
	strcpy(node[i++].var.Format, "%name%: %s");

	node[i].pHeadNode	= (UDINT)&node[P_PARAM_WF];
	node[i].Type = N_EDIT;
	node[i].MinUserLevel = 5;
	node[i].var.Type = T_SCALED;
	node[i].var.Var1ID = parWF_SpeedFinal;
	//strcpy(node[i++].var.Format, "WF FIN SP %s");
	strcpy(node[i++].var.Format, "%name%: %s");

	node[i].pHeadNode	= (UDINT)&node[P_PARAM_WF];
	node[i].Type = N_EDIT;
	node[i].MinUserLevel = 5;
	node[i].var.Type = T_SCALED;
	node[i].var.Var1ID = parWF_RetractSpeed;
	//strcpy(node[i++].var.Format, "WF RET SP %s");
	strcpy(node[i++].var.Format, "%name%: %s");

	node[i].pHeadNode	= (UDINT)&node[P_PARAM_WF];
	node[i].Type = N_EDIT;
	node[i].MinUserLevel = 5;
	node[i].var.Type = T_SCALED;
	node[i].var.Var1ID = parWF_RetracDist;
	//strcpy(node[i++].var.Format, "WF UP LEN %s");
	strcpy(node[i++].var.Format, "%name%: %s");

	node[i].pHeadNode	= (UDINT)&node[P_PARAM_WF];
	node[i].Type = N_EDIT;
	node[i].MinUserLevel = 5;
	node[i].var.Type = T_SCALED;
	node[i].var.Var1ID = parWF_RampUpdate;
	//strcpy(node[i++].var.Format, "RampUpdate: %s");
	strcpy(node[i++].var.Format, "%name%: %s");

	node[i].pHeadNode	= (UDINT)&node[P_PARAM_WF];
	node[i].Type = N_EDIT;
	node[i].MinUserLevel = 5;
	node[i].var.Type = T_ENUM;
	node[i].var.Var1ID = parENUM_WF_AUX;
	strcpy(node[i++].var.Format, "%name%: %s");

	/*
	node[i].pHeadNode	= (UDINT)&node[P_PARAM_WF];
	node[i].Type = N_EDIT;
	node[i].MinUserLevel = 5;
	node[i].var.Type = T_SCALED;
	node[i].var.Var1ID = parWF_Boost1SP;
	//strcpy(node[i++].var.Format, "Boost1: %s");
	strcpy(node[i++].var.Format, "%name%: %s");

	node[i].pHeadNode	= (UDINT)&node[P_PARAM_WF];
	node[i].Type = N_EDIT;
	node[i].MinUserLevel = 5;
	node[i].var.Type = T_SCALED;
	node[i].var.Var1ID = parWF_Boost2SP;
	//strcpy(node[i++].var.Format, "Boost2: %s");
	strcpy(node[i++].var.Format, "%name%: %s");
	*/

	node[i].pHeadNode	= (UDINT)&node[P_PARAM_WF];
	node[i].Type = N_EDIT;
	node[i].MinUserLevel = 5;
	node[i].var.Type = T_SCALED;
	node[i].var.Var1ID = parWF_JogSpeed;
	//strcpy(node[i++].var.Format, "Jog Vel.: %s");
	strcpy(node[i++].var.Format, "%name%: %s");

	node[i].pHeadNode	= (UDINT)&node[P_PARAM_WF];
	node[i].Type = N_EDIT;
	node[i].MinUserLevel = 5;
	node[i].var.Type = T_SCALED;
	node[i].var.Var1ID = parWF_JogSpeedDirCntrl;
	//strcpy(node[i++].var.Format, "Jog Cntrl: %s");
	strcpy(node[i++].var.Format, "%name%: %s");

	node[i].pHeadNode	= (UDINT)&node[P_PARAM_WF];
	node[i].Type = N_EDIT;
	node[i].MinUserLevel = 5;
	node[i].var.Type = T_SCALED;
	node[i].var.Var1ID = parWF_CalibVel1;
	//strcpy(node[i++].var.Format, "Cal.Vel1: %s");
	strcpy(node[i++].var.Format, "%name%: %s");

	node[i].pHeadNode	= (UDINT)&node[P_PARAM_WF];
	node[i].Type = N_EDIT;
	node[i].MinUserLevel = 5;
	node[i].var.Type = T_SCALED;
	node[i].var.Var1ID = parWF_CalibVel2;
	//strcpy(node[i++].var.Format, "Cal.Vel2: %s");
	strcpy(node[i++].var.Format, "%name%: %s");

	node[i].pHeadNode	= (UDINT)&node[P_PARAM_WF];
	node[i].Type = N_SCROLL + N_NO_PREFIX;
	node[i].MinUserLevel = 5;
	strcpy(node[i++].var.Format, "**** CALCULATED ****");

	node[i].pHeadNode	= (UDINT)&node[P_PARAM_WF];
	node[i].Type = N_EDIT;
	node[i].MinUserLevel = 5;
	node[i].var.Type = T_SCALED;
	node[i].var.Var1ID = parWF_StartDly;
	//strcpy(node[i++].var.Format, "WF DLY %s");
	strcpy(node[i++].var.Format, "%name%: %s");

	node[i].pHeadNode	= (UDINT)&node[P_PARAM_WF];
	node[i].Type = N_EDIT;
	node[i].MinUserLevel = 5;
	node[i].var.Type = T_SCALED;
	node[i].var.Var1ID = parWF_RampUp;
	//strcpy(node[i++].var.Format, "WF UPSLOP %s");
	strcpy(node[i++].var.Format, "%name%: %s");

	node[i].pHeadNode	= (UDINT)&node[P_PARAM_WF];
	node[i].Type = N_EDIT;
	node[i].MinUserLevel = 5;
	node[i].var.Type = T_SCALED;
	node[i].var.Var1ID = parWF_StopDly;
	//strcpy(node[i++].var.Format, "WF DS DLY %s");
	strcpy(node[i++].var.Format, "%name%: %s");

	node[i].pHeadNode	= (UDINT)&node[P_PARAM_WF];
	node[i].Type = N_EDIT;
	node[i].MinUserLevel = 5;
	node[i].var.Type = T_SCALED;
	node[i].var.Var1ID = parWF_RampDwn;
	//strcpy(node[i++].var.Format, "WF DWNSLP %s");
	strcpy(node[i++].var.Format, "%name%: %s");

	node[i].pHeadNode	= (UDINT)&node[P_PARAM_WF];
	node[i].Type = N_EDIT;
	node[i].MinUserLevel = 5;
	node[i].var.Type = T_SCALED;
	node[i].var.Var1ID = parWF_RetractDly;
	//strcpy(node[i++].var.Format, "WFRET DLY %s");
	strcpy(node[i++].var.Format, "%name%: %s");

	/** P_PARAM_AVC **/
	i = P_PARAM_AVC;			h=varSTRING_HMI_0;
	SetPageDict(&cfg->PagesDict[n++] , P_PARAM_AVC , "P_PARAM_AVC");

	node[i].pHeadNode	= (UDINT)&node[P_PARAM_AVC];
	node[i].Type = N_JUMP;
	node[i].JumpLineID = 0;
	node[i].pJumpNode = (UDINT)&node[P_PARAM];
	strcpy(node[i++].var.Format, "Return ");

	node[i].pHeadNode	= (UDINT)&node[P_PARAM_AVC];
	node[i].Type = N_EDIT;
	node[i].MinUserLevel = 5;
	node[i].var.Type = T_SCALED;
	node[i].var.Var1ID = parAVC_VoltSP;
	//strcpy(node[i++].var.Format, "PRI VOLTS %s");
	strcpy(node[i++].var.Format, "%name%: %s");

	node[i].pHeadNode	= (UDINT)&node[P_PARAM_AVC];
	node[i].Type = N_EDIT;
	node[i].MinUserLevel = 5;
	node[i].var.Type = T_SCALED;
	node[i].var.Var1ID = parAVC_VoltInSP;
	//strcpy(node[i++].var.Format, "PRI IN VOLTS %s");
	strcpy(node[i++].var.Format, "%name%: %s");

	node[i].pHeadNode	= (UDINT)&node[P_PARAM_AVC];
	node[i].Type = N_EDIT;
	node[i].MinUserLevel = 5;
	node[i].var.Type = T_SCALED;
	node[i].var.Var1ID = parAVC_VoltOutSP;
	//strcpy(node[i++].var.Format, "PRI OUT VOLTS %s");
	strcpy(node[i++].var.Format, "%name%: %s");

	node[i].pHeadNode	= (UDINT)&node[P_PARAM_AVC];
	node[i].Type = N_EDIT;
	node[i].MinUserLevel = 5;
	node[i].var.Type = T_SCALED;
	node[i].var.Var1ID = parAVC_VoltBackSP;
	//strcpy(node[i++].var.Format, "BACK VOLTS %s");
	strcpy(node[i++].var.Format, "%name%: %s");

	node[i].pHeadNode	= (UDINT)&node[P_PARAM_AVC];
	node[i].Type = N_EDIT;
	node[i].MinUserLevel = 5;
	node[i].var.Type = T_ENUM;
	node[i].var.Var1ID = parENUM_AVC_Mode;
	//strcpy(node[i++].var.Format, "Mode: %s");
	strcpy(node[i++].var.Format, "%name%: %s");

	node[i].pHeadNode 	= (UDINT)&node[P_PARAM_AVC];
	node[i].Type = N_SCROLL + N_NO_PREFIX;
	node[i].MinUserLevel = 5;
	strcpy(node[i++].var.Format, "** ARC Start/Stop **");

	node[i].pHeadNode	= (UDINT)&node[P_PARAM_AVC];
	node[i].Type = N_EDIT;
	node[i].MinUserLevel = 5;
	node[i].var.Type = T_SCALED;
	node[i].var.Var1ID = parAVC_TouchVolt;
	//strcpy(node[i++].var.Format, "TOUCH V %s");
	strcpy(node[i++].var.Format, "%name%: %s");

	node[i].pHeadNode	= (UDINT)&node[P_PARAM_AVC];
	node[i].Type = N_EDIT;
	node[i].MinUserLevel = 5;
	node[i].var.Type = T_SCALED;
	node[i].var.Var1ID = parAVC_VoltInit;
	//strcpy(node[i++].var.Format, "AVC INI V %s");
	strcpy(node[i++].var.Format, "%name%: %s");

	node[i].pHeadNode	= (UDINT)&node[P_PARAM_AVC];
	node[i].Type = N_EDIT;
	node[i].MinUserLevel = 5;
	node[i].var.Type = T_SCALED;
	node[i].var.Var1ID = parAVC_TouchVel;
	//strcpy(node[i++].var.Format, "AVC SRI %s");
	strcpy(node[i++].var.Format, "%name%: %s");

	node[i].pHeadNode	= (UDINT)&node[P_PARAM_AVC];
	node[i].Type = N_EDIT;
	node[i].MinUserLevel = 5;
	node[i].var.Type = T_SCALED;
	node[i].var.Var1ID = parAVC_KissTm;
	//strcpy(node[i++].var.Format, "Touch Time %s");
	strcpy(node[i++].var.Format, "%name%: %s");

	node[i].pHeadNode	= (UDINT)&node[P_PARAM_AVC];
	node[i].Type = N_EDIT;
	node[i].MinUserLevel = 5;
	node[i].var.Type = T_SCALED;
	node[i].var.Var1ID = parAVC_ToSPVel;
	//strcpy(node[i++].var.Format, "AVC LU SP %s");
	strcpy(node[i++].var.Format, "%name%: %s");

	node[i].pHeadNode	= (UDINT)&node[P_PARAM_AVC];
	node[i].Type = N_EDIT;
	node[i].MinUserLevel = 5;
	node[i].var.Type = T_SCALED;
	node[i].var.Var1ID = parAVC_LU_TM;
	//strcpy(node[i++].var.Format, "AVC LU TM %s");
	strcpy(node[i++].var.Format, "%name%: %s");

	node[i].pHeadNode	= (UDINT)&node[P_PARAM_AVC];
	node[i].Type = N_EDIT;
	node[i].MinUserLevel = 5;
	node[i].var.Type = T_SCALED;
	node[i].var.Var1ID = parAVC_VoltFinal;
	//strcpy(node[i++].var.Format, "FIN VOLTS %s");
	strcpy(node[i++].var.Format, "%name%: %s");

	node[i].pHeadNode	= (UDINT)&node[P_PARAM_AVC];
	node[i].Type = N_EDIT;
	node[i].MinUserLevel = 5;
	node[i].var.Type = T_SCALED;
	node[i].var.Var1ID = parAVC_GoBackTm;
	//strcpy(node[i++].var.Format, "AVC UP TM %s");
	strcpy(node[i++].var.Format, "%name%: %s");

	node[i].pHeadNode	= (UDINT)&node[P_PARAM_AVC];
	node[i].Type = N_EDIT;
	node[i].MinUserLevel = 5;
	node[i].var.Type = T_SCALED;
	node[i].var.Var1ID = parAVC_LiftSpeedDirCntrl;
	//strcpy(node[i++].var.Format, "AVC UP SP %s");
	strcpy(node[i++].var.Format, "%name%: %s");

	node[i].pHeadNode	= (UDINT)&node[P_PARAM_AVC];
	node[i].Type = N_EDIT;
	node[i].MinUserLevel = 5;
	node[i].var.Type = T_SCALED;
	node[i].var.Var1ID = parAVC_TouchTm;
	//strcpy(node[i++].var.Format, "Touch TMO: %s");
	strcpy(node[i++].var.Format, "%name%: %s");

	node[i].pHeadNode	= (UDINT)&node[P_PARAM_AVC];
	node[i].Type = N_EDIT;
	node[i].MinUserLevel = 5;
	node[i].var.Type = T_SCALED;
	node[i].var.Var1ID = parAVC_TRetractTm;
	//strcpy(node[i++].var.Format, "Retract: %s");
	strcpy(node[i++].var.Format, "%name%: %s");

	node[i].pHeadNode	= (UDINT)&node[P_PARAM_AVC];
	node[i].Type = N_EDIT;
	node[i].MinUserLevel = 5;
	node[i].var.Type = T_SCALED;
	node[i].var.Var1ID = parAVC_TouchRepeat;
	//strcpy(node[i++].var.Format, "Repeat Cnt: %s");
	strcpy(node[i++].var.Format, "%name%: %s");

	/*
	node[i].pHeadNode 	= (UDINT)&node[P_PARAM_AVC];
	node[i].Type = N_SCROLL + N_NO_PREFIX;
	node[i].MinUserLevel = 5;
	strcpy(node[i++].var.Format, "******* MSC. *******");
	*/

	node[i].pHeadNode	= (UDINT)&node[P_PARAM_AVC];
	node[i].Type = N_EDIT;
	node[i].MinUserLevel = 5;
	node[i].var.Type = T_SCALED;
	node[i].var.Var1ID = parAVC_StartDly;
	//strcpy(node[i++].var.Format, "V UPS DLY %s");
	strcpy(node[i++].var.Format, "%name%: %s");

	node[i].pHeadNode	= (UDINT)&node[P_PARAM_AVC];
	node[i].Type = N_EDIT;
	node[i].MinUserLevel = 5;
	node[i].var.Type = T_SCALED;
	node[i].var.Var1ID = parAVC_VSPTmOut;
	//strcpy(node[i++].var.Format, "Init Volt Tmo: %s");
	strcpy(node[i++].var.Format, "%name%: %s");

	node[i].pHeadNode	= (UDINT)&node[P_PARAM_AVC];
	node[i].Type = N_EDIT;
	node[i].MinUserLevel = 5;
	node[i].var.Type = T_SCALED;
	node[i].var.Var1ID = parAVC_MaxVoltError;
	//strcpy(node[i++].var.Format, "Max Volt Err: %s");
	strcpy(node[i++].var.Format, "%name%: %s");

	node[i].pHeadNode	= (UDINT)&node[P_PARAM_AVC];
	node[i].Type = N_EDIT;
	node[i].MinUserLevel = 5;
	node[i].var.Type = T_SCALED;
	node[i].var.Var1ID = parAVC_JogSpeedDirCntrl;
	//strcpy(node[i++].var.Format, "Jog Cntrl: %s");
	strcpy(node[i++].var.Format, "%name%: %s");

	/*
	node[i].pHeadNode	= (UDINT)&node[P_PARAM_AVC];
	node[i].Type = N_EDIT;
	node[i].MinUserLevel = 5;
	node[i].var.Type = T_SCALED;
	node[i].var.Var1ID = parAVC_Limits_Mask_Tm;
	strcpy(node[i++].var.Format, "Lim Filt: %s");
	*/

	node[i].pHeadNode	= (UDINT)&node[P_PARAM_AVC];
	node[i].Type = N_EDIT;
	node[i].MinUserLevel = 5;
	node[i].var.Type = T_SCALED;
	node[i].var.Var1ID = parAVC_FbkFilter;
	//strcpy(node[i++].var.Format, "Fbk Filtr: %s");
	strcpy(node[i++].var.Format, "%name%: %s");

	node[i].pHeadNode	= (UDINT)&node[P_PARAM_AVC];
	node[i].Type = N_EDIT;
	node[i].MinUserLevel = 5;
	node[i].var.Type = T_SCALED;
	node[i].var.Var1ID = parAVC_KPP;
	//strcpy(node[i++].var.Format, "KPP: %s");
	strcpy(node[i++].var.Format, "%name%: %s");

	node[i].pHeadNode	= (UDINT)&node[P_PARAM_AVC];
	node[i].Type = N_EDIT;
	node[i].MinUserLevel = 5;
	node[i].var.Type = T_SCALED;
	node[i].var.Var1ID = parAVC_KIP;
	//strcpy(node[i++].var.Format, "KIP: %s");
	strcpy(node[i++].var.Format, "%name%: %s");

	node[i].pHeadNode	= (UDINT)&node[P_PARAM_AVC];
	node[i].Type = N_EDIT;
	node[i].MinUserLevel = 5;
	node[i].var.Type = T_SCALED;
	node[i].var.Var1ID = parAVC_DB_Window;
	//strcpy(node[i++].var.Format, "DB Window: %s");
	strcpy(node[i++].var.Format, "%name%: %s");

	node[i].pHeadNode	= (UDINT)&node[P_PARAM_AVC];
	node[i].Type = N_EDIT;
	node[i].MinUserLevel = 5;
	node[i].var.Type = T_SCALED;
	node[i].var.Var1ID = parAVC_BB_Vel;
	//strcpy(node[i++].var.Format, "BB Speed: %s");
	strcpy(node[i++].var.Format, "%name%: %s");

	node[i].pHeadNode	= (UDINT)&node[P_PARAM_AVC];
	node[i].Type = N_EDIT;
	node[i].MinUserLevel = 5;
	node[i].var.Type = T_SCALED;
	node[i].var.Var1ID = parAVC_BB_Gain;
	//strcpy(node[i++].var.Format, "BB Gain: %s");
	strcpy(node[i++].var.Format, "%name%: %s");

	node[i].pHeadNode	= (UDINT)&node[P_PARAM_AVC];
	node[i].Type = N_EDIT;
	node[i].MinUserLevel = 5;
	node[i].var.Type = T_SCALED;
	node[i].var.Var1ID = parAVC_BB_Integr;
	strcpy(node[i++].var.Format, "%name%: %s");

	node[i].pHeadNode	= (UDINT)&node[P_PARAM_AVC];
	node[i].Type = N_SCROLL + N_NO_PREFIX;
	node[i].MinUserLevel = 5;
	strcpy(node[i++].var.Format, "**** CALCULATED ****");

	node[i].pHeadNode	= (UDINT)&node[P_PARAM_AVC];
	node[i].Type = N_EDIT;
	node[i].MinUserLevel = 5;
	node[i].var.Type = T_SCALED;
	node[i].var.Var1ID = parAVC_Upslope;
	//strcpy(node[i++].var.Format, "V UPSLOPE %s");
	strcpy(node[i++].var.Format, "%name%: %s");

	node[i].pHeadNode	= (UDINT)&node[P_PARAM_AVC];
	node[i].Type = N_EDIT;
	node[i].MinUserLevel = 5;
	node[i].var.Type = T_SCALED;
	node[i].var.Var1ID = parAVC_StopDly;
	//strcpy(node[i++].var.Format, "V DS DLY %s");
	strcpy(node[i++].var.Format, "%name%: %s");

	node[i].pHeadNode	= (UDINT)&node[P_PARAM_AVC];
	node[i].Type = N_EDIT;
	node[i].MinUserLevel = 5;
	node[i].var.Type = T_SCALED;
	node[i].var.Var1ID = parAVC_DownSlope;
	//strcpy(node[i++].var.Format, "V DWNSLOP %s");
	strcpy(node[i++].var.Format, "%name%: %s");

	node[i].pHeadNode	= (UDINT)&node[P_PARAM_AVC];
	node[i].Type = N_EDIT;
	node[i].MinUserLevel = 5;
	node[i].var.Type = T_SCALED;
	node[i].var.Var1ID = parAVC_HoldTm;
	//strcpy(node[i++].var.Format, "AVCUP DLY %s");
	strcpy(node[i++].var.Format, "%name%: %s");

	/** P_PARAM_TIG **/
	i = P_PARAM_TIG;			h=varSTRING_HMI_0;
	SetPageDict(&cfg->PagesDict[n++] , P_PARAM_TIG , "P_PARAM_TIG");

	node[i].pHeadNode	= (UDINT)&node[P_PARAM_TIG];
	node[i].Type = N_JUMP;
	node[i].JumpLineID = 0;
	node[i].pJumpNode = (UDINT)&node[P_PARAM];
	strcpy(node[i++].var.Format, "Return ");

	node[i].pHeadNode	= (UDINT)&node[P_PARAM_TIG];
	node[i].Type = N_EDIT;
	node[i].MinUserLevel = 5;
	node[i].var.Type = T_SCALED;
	node[i].var.Var1ID = parTIG_AmpSP;
	//strcpy(node[i++].var.Format, "PRI AMPS %s");
	strcpy(node[i++].var.Format, "%name%: %s");

	node[i].pHeadNode	= (UDINT)&node[P_PARAM_TIG];
	node[i].Type = N_EDIT;
	node[i].MinUserLevel = 5;
	node[i].var.Type = T_SCALED;
	node[i].var.Var1ID = parTIG_AmpInSP;
	//strcpy(node[i++].var.Format, "PRI IN AMPS %s");
	strcpy(node[i++].var.Format, "%name%: %s");

	node[i].pHeadNode	= (UDINT)&node[P_PARAM_TIG];
	node[i].Type = N_EDIT;
	node[i].MinUserLevel = 5;
	node[i].var.Type = T_SCALED;
	node[i].var.Var1ID = parTIG_AmpOutSP;
	//strcpy(node[i++].var.Format, "PRI OUT AMPS %s");
	strcpy(node[i++].var.Format, "%name%: %s");

	node[i].pHeadNode	= (UDINT)&node[P_PARAM_TIG];
	node[i].Type = N_EDIT;
	node[i].MinUserLevel = 5;
	node[i].var.Type = T_SCALED;
	node[i].var.Var1ID = parTIG_BackAmp;
	//strcpy(node[i++].var.Format, "BKG AMPS %s");
	strcpy(node[i++].var.Format, "%name%: %s");

	node[i].pHeadNode	= (UDINT)&node[P_PARAM_TIG];
	node[i].Type = N_EDIT;
	node[i].MinUserLevel = 5;
	node[i].var.Type = T_SCALED;
	node[i].var.Var1ID = parTIG_PulseFreq;
	//strcpy(node[i++].var.Format, "Pulse Freq. %s");
	strcpy(node[i++].var.Format, "%name%: %s");

	node[i].pHeadNode	= (UDINT)&node[P_PARAM_TIG];
	node[i].Type = N_EDIT;
	node[i].MinUserLevel = 5;
	node[i].var.Type = T_SCALED;
	node[i].var.Var1ID = parTIG_PulseWidth;
	//strcpy(node[i++].var.Format, "Pulse Width %s");
	strcpy(node[i++].var.Format, "%name%: %s");

	node[i].pHeadNode 	= (UDINT)&node[P_PARAM_TIG];
	node[i].Type = N_EDIT;
	node[i].MinUserLevel = 5;
	node[i].var.Type = T_ENUM;
	node[i].var.Var1ID = parENUM_TIG_Mode;
	//strcpy(node[i++].var.Format, "Mode: %s");
	strcpy(node[i++].var.Format, "%name%: %s");

	node[i].pHeadNode 	= (UDINT)&node[P_PARAM_TIG];
	node[i].Type = N_SCROLL + N_NO_PREFIX;
	node[i].MinUserLevel = 5;
	strcpy(node[i++].var.Format, "******* MSC. *******");

	node[i].pHeadNode	= (UDINT)&node[P_PARAM_TIG];
	node[i].Type = N_EDIT;
	node[i].MinUserLevel = 5;
	node[i].var.Type = T_SCALED;
	node[i].var.Var1ID = parTIG_StartAmp;
	//strcpy(node[i++].var.Format, "INI AMPS %s");
	strcpy(node[i++].var.Format, "%name%: %s");

	node[i].pHeadNode	= (UDINT)&node[P_PARAM_TIG];
	node[i].Type = N_EDIT;
	node[i].MinUserLevel = 5;
	node[i].var.Type = T_SCALED;
	node[i].var.Var1ID = parTIG_EndAmp;
	//strcpy(node[i++].var.Format, "FIN AMPS %s");
	strcpy(node[i++].var.Format, "%name%: %s");

	node[i].pHeadNode	= (UDINT)&node[P_PARAM_TIG];
	node[i].Type = N_EDIT;
	node[i].MinUserLevel = USER_MANAGER;
	node[i].var.Type = T_SCALED;
	node[i].var.Var1ID = parTIG_AmpSP_Boost;
	//strcpy(node[i++].var.Format, "Amp Boost: %s");
	strcpy(node[i++].var.Format, "%name%: %s");

	node[i].pHeadNode 	= (UDINT)&node[P_PARAM_TIG];
	node[i].Type = N_EDIT;
	node[i].MinUserLevel = 5;
	node[i].var.Type = T_ENUM;
	node[i].var.Var1ID = parENUM_ARCLINK_MODE;
	//strcpy(node[i++].var.Format, "ArcLink: %s");
	strcpy(node[i++].var.Format, "%name%: %s");

	node[i].pHeadNode	= (UDINT)&node[P_PARAM_TIG];
	node[i].Type = N_EDIT;
	node[i].MinUserLevel = USER_MANAGER;
	node[i].var.Type = T_SCALED;
	node[i].var.Var1ID = parTIG_CalibAmp1;
	//strcpy(node[i++].var.Format, "Cal. Amp1: %s");
	strcpy(node[i++].var.Format, "%name%: %s");

	node[i].pHeadNode	= (UDINT)&node[P_PARAM_TIG];
	node[i].Type = N_EDIT;
	node[i].MinUserLevel = USER_MANAGER;
	node[i].var.Type = T_SCALED;
	node[i].var.Var1ID = parTIG_CalibAmp2;
	//strcpy(node[i++].var.Format, "Cal. Amp2: %s");
	strcpy(node[i++].var.Format, "%name%: %s");

	node[i].pHeadNode	= (UDINT)&node[P_PARAM_TIG];
	node[i].Type = N_SCROLL + N_NO_PREFIX;
	node[i].MinUserLevel = 5;
	strcpy(node[i++].var.Format, "**** CALCULATED ****");

	node[i].pHeadNode	= (UDINT)&node[P_PARAM_TIG];
	node[i].Type = N_EDIT;
	node[i].MinUserLevel = 5;
	node[i].var.Type = T_SCALED;
	node[i].var.Var1ID = parTIG_StartDly;
	//strcpy(node[i++].var.Format, "I DLY %s");
	strcpy(node[i++].var.Format, "%name%: %s");

	node[i].pHeadNode	= (UDINT)&node[P_PARAM_TIG];
	node[i].Type = N_EDIT;
	node[i].MinUserLevel = 5;
	node[i].var.Type = T_SCALED;
	node[i].var.Var1ID = parTIG_RampUp;
	//strcpy(node[i++].var.Format, "I UPSLOPE %s");
	strcpy(node[i++].var.Format, "%name%: %s");

	node[i].pHeadNode	= (UDINT)&node[P_PARAM_TIG];
	node[i].Type = N_EDIT;
	node[i].MinUserLevel = 5;
	node[i].var.Type = T_SCALED;
	node[i].var.Var1ID = parTIG_StopDly;
	//strcpy(node[i++].var.Format, "I DS DLY %s");
	strcpy(node[i++].var.Format, "%name%: %s");

	node[i].pHeadNode	= (UDINT)&node[P_PARAM_TIG];
	node[i].Type = N_EDIT;
	node[i].MinUserLevel = 5;
	node[i].var.Type = T_SCALED;
	node[i].var.Var1ID = parTIG_RampDwn;
	//strcpy(node[i++].var.Format, "I DOWNSLOP %s");
	strcpy(node[i++].var.Format, "%name%: %s");

	/** P_PARAM_HW **/
	i = P_PARAM_HW;			h=varSTRING_HMI_0;
	SetPageDict(&cfg->PagesDict[n++] , P_PARAM_HW , "P_PARAM_HW");

	node[i].pHeadNode	= (UDINT)&node[P_PARAM_HW];
	node[i].Type = N_JUMP;
	node[i].JumpLineID = 0;
	node[i].pJumpNode = (UDINT)&node[P_PARAM];
	strcpy(node[i++].var.Format, "Return ");

	node[i].pHeadNode	= (UDINT)&node[P_PARAM_HW];
	node[i].Type = N_EDIT;
	node[i].MinUserLevel = 5;
	node[i].var.Type = T_SCALED;
	node[i].var.Var1ID = parHW_AmpSP;
	//strcpy(node[i++].var.Format, "HW PRI A %s");
	strcpy(node[i++].var.Format, "%name%: %s");

	node[i].pHeadNode 	= (UDINT)&node[P_PARAM_HW];
	node[i].Type = N_SCROLL + N_NO_PREFIX;
	node[i].MinUserLevel = 5;
	strcpy(node[i++].var.Format, "******* MSC. *******");

	node[i].pHeadNode	= (UDINT)&node[P_PARAM_HW];
	node[i].Type = N_EDIT;
	node[i].MinUserLevel = 5;
	node[i].var.Type = T_SCALED;
	node[i].var.Var1ID = parHW_StartAmp;
	//strcpy(node[i++].var.Format, "HW INI A %s");
	strcpy(node[i++].var.Format, "%name%: %s");

	node[i].pHeadNode	= (UDINT)&node[P_PARAM_HW];
	node[i].Type = N_EDIT;
	node[i].MinUserLevel = 5;
	node[i].var.Type = T_SCALED;
	node[i].var.Var1ID = parHW_EndAmp;
	//strcpy(node[i++].var.Format, "HW FIN A %s");
	strcpy(node[i++].var.Format, "%name%: %s");

	node[i].pHeadNode	= (UDINT)&node[P_PARAM_HW];
	node[i].Type = N_EDIT;
	node[i].MinUserLevel = 5;
	node[i].var.Type = T_SCALED;
	node[i].var.Var1ID = parHW_VoltSP;
	//strcpy(node[i++].var.Format, "Prim Volt: %s");
	strcpy(node[i++].var.Format, "%name%: %s");

	node[i].pHeadNode	= (UDINT)&node[P_PARAM_HW];
	node[i].Type = N_EDIT;
	node[i].MinUserLevel = USER_MANAGER;
	node[i].var.Type = T_SCALED;
	node[i].var.Var1ID = parHW_AmpSP_Boost;
	//strcpy(node[i++].var.Format, "Amp Boost: %s");
	strcpy(node[i++].var.Format, "%name%: %s");

	node[i].pHeadNode	= (UDINT)&node[P_PARAM_HW];
	node[i].Type = N_EDIT;
	node[i].MinUserLevel = 5;
	node[i].var.Type = T_SCALED;
	node[i].var.Var1ID = parTIG_CalibAmp1;
	//strcpy(node[i++].var.Format, "Cal. Amp1: %s");
	strcpy(node[i++].var.Format, "%name%: %s");

	node[i].pHeadNode	= (UDINT)&node[P_PARAM_HW];
	node[i].Type = N_EDIT;
	node[i].MinUserLevel = 5;
	node[i].var.Type = T_SCALED;
	node[i].var.Var1ID = parTIG_CalibAmp2;
	//strcpy(node[i++].var.Format, "Cal. Amp2: %s");
	strcpy(node[i++].var.Format, "%name%: %s");

	node[i].pHeadNode	= (UDINT)&node[P_PARAM_HW];
	node[i].Type = N_SCROLL + N_NO_PREFIX;
	node[i].MinUserLevel = 5;
	strcpy(node[i++].var.Format, "**** CALCULATED ****");

	node[i].pHeadNode	= (UDINT)&node[P_PARAM_HW];
	node[i].Type = N_EDIT;
	node[i].MinUserLevel = 5;
	node[i].var.Type = T_SCALED;
	node[i].var.Var1ID = parHW_RampUpDly;
	//strcpy(node[i++].var.Format, "HW US DLY %s");
	strcpy(node[i++].var.Format, "%name%: %s");

	node[i].pHeadNode	= (UDINT)&node[P_PARAM_HW];
	node[i].Type = N_EDIT;
	node[i].MinUserLevel = 5;
	node[i].var.Type = T_SCALED;
	node[i].var.Var1ID = parHW_RampUp;
	//strcpy(node[i++].var.Format, "HW UPSLOP %s");
	strcpy(node[i++].var.Format, "%name%: %s");

	node[i].pHeadNode	= (UDINT)&node[P_PARAM_HW];
	node[i].Type = N_EDIT;
	node[i].MinUserLevel = 5;
	node[i].var.Type = T_SCALED;
	node[i].var.Var1ID = parHW_RampDwnDly;
	//strcpy(node[i++].var.Format, "HW DS DLY %s");
	strcpy(node[i++].var.Format, "%name%: %s");

	node[i].pHeadNode	= (UDINT)&node[P_PARAM_HW];
	node[i].Type = N_EDIT;
	node[i].MinUserLevel = 5;
	node[i].var.Type = T_SCALED;
	node[i].var.Var1ID = parHW_RampDwn;
	//strcpy(node[i++].var.Format, "HW DWNSLOP %s");
	strcpy(node[i++].var.Format, "%name%: %s");

	/** P_PARAM_BOOSTS **/
	i = P_PARAM_BOOSTS;			h=varSTRING_HMI_0;
	SetPageDict(&cfg->PagesDict[n++] , P_PARAM_BOOSTS , "P_PARAM_BOOSTS");

	node[i].pHeadNode	= (UDINT)&node[P_PARAM_BOOSTS];
	node[i].Type = N_JUMP;
	node[i].JumpLineID = 0;
	node[i].pJumpNode = (UDINT)&node[P_MENU];
	strcpy(node[i++].var.Format, "Return ");

	node[i].pHeadNode	= (UDINT)&node[P_PARAM_BOOSTS];
	node[i].Type = N_SCROLL;
	strcpy(node[i++].var.Format, " *BOOST 1 - UP Key* ");

	node[i].pHeadNode 	= (UDINT)&node[P_PARAM_BOOSTS];
	node[i].Type = N_EDIT;
	node[i].MinUserLevel = 5;
	node[i].var.Type = T_SCALED;
	node[i].var.Var1ID = parTIG_Boost1;
	//strcpy(node[i++].var.Format, "T PRI SP %s");
	strcpy(node[i++].var.Format, "%name%: %s");

	node[i].pHeadNode 	= (UDINT)&node[P_PARAM_BOOSTS];
	node[i].Type = N_EDIT;
	node[i].MinUserLevel = 5;
	node[i].var.Type = T_SCALED;
	node[i].var.Var1ID = parAVC_Boost1;
	//strcpy(node[i++].var.Format, "T PRI SP %s");
	strcpy(node[i++].var.Format, "%name%: %s");

	node[i].pHeadNode 	= (UDINT)&node[P_PARAM_BOOSTS];
	node[i].Type = N_EDIT;
	node[i].MinUserLevel = 5;
	node[i].var.Type = T_SCALED;
	node[i].var.Var1ID = parTVL_Boost1;
	//strcpy(node[i++].var.Format, "T PRI SP %s");
	strcpy(node[i++].var.Format, "%name%: %s");

	node[i].pHeadNode 	= (UDINT)&node[P_PARAM_BOOSTS];
	node[i].Type = N_EDIT;
	node[i].MinUserLevel = 5;
	node[i].var.Type = T_SCALED;
	node[i].var.Var1ID = parWF_Boost1SP;
	//strcpy(node[i++].var.Format, "T PRI SP %s");
	strcpy(node[i++].var.Format, "%name%: %s");

	node[i].pHeadNode	= (UDINT)&node[P_PARAM_BOOSTS];
	node[i].Type = N_EDIT;
	node[i].MinUserLevel = 5;
	node[i].var.Type = T_SCALED;
	node[i].var.Var1ID = parWP_Boost1SP;
	//strcpy(node[i++].var.Format, "T PRI SP %s");
	strcpy(node[i++].var.Format, "%name%: %s");

	node[i].pHeadNode	= (UDINT)&node[P_PARAM_BOOSTS];
	node[i].Type = N_SCROLL;
	strcpy(node[i++].var.Format, " *BOOST 2 - Down Key* ");

	node[i].pHeadNode 	= (UDINT)&node[P_PARAM_BOOSTS];
	node[i].Type = N_EDIT;
	node[i].MinUserLevel = 5;
	node[i].var.Type = T_SCALED;
	node[i].var.Var1ID = parTIG_Boost2;
	//strcpy(node[i++].var.Format, "T PRI SP %s");
	strcpy(node[i++].var.Format, "%name%: %s");

	node[i].pHeadNode	= (UDINT)&node[P_PARAM_BOOSTS];
	node[i].Type = N_EDIT;
	node[i].MinUserLevel = 5;
	node[i].var.Type = T_SCALED;
	node[i].var.Var1ID = parAVC_Boost2;
	//strcpy(node[i++].var.Format, "T PRI SP %s");
	strcpy(node[i++].var.Format, "%name%: %s");

	node[i].pHeadNode	= (UDINT)&node[P_PARAM_BOOSTS];
	node[i].Type = N_EDIT;
	node[i].MinUserLevel = 5;
	node[i].var.Type = T_SCALED;
	node[i].var.Var1ID = parTVL_Boost2;
	//strcpy(node[i++].var.Format, "T PRI SP %s");
	strcpy(node[i++].var.Format, "%name%: %s");

	node[i].pHeadNode 	= (UDINT)&node[P_PARAM_BOOSTS];
	node[i].Type = N_EDIT;
	node[i].MinUserLevel = 5;
	node[i].var.Type = T_SCALED;
	node[i].var.Var1ID = parWF_Boost2SP;
	//strcpy(node[i++].var.Format, "T PRI SP %s");
	strcpy(node[i++].var.Format, "%name%: %s");

	node[i].pHeadNode	= (UDINT)&node[P_PARAM_BOOSTS];
	node[i].Type = N_EDIT;
	node[i].MinUserLevel = 5;
	node[i].var.Type = T_SCALED;
	node[i].var.Var1ID = parWP_Boost2SP;
	//strcpy(node[i++].var.Format, "T PRI SP %s");
	strcpy(node[i++].var.Format, "%name%: %s");

	/** P_PARAM_CONTIN_WELD **/
	i = P_PARAM_CONTIN_WELD;			h=varSTRING_HMI_0;
	SetPageDict(&cfg->PagesDict[n++] , P_PARAM_CONTIN_WELD , "P_PARAM_CONTIN_WELD");

	node[i].pHeadNode	= (UDINT)&node[P_PARAM_CONTIN_WELD];
	node[i].Type = N_JUMP;
	node[i].JumpLineID = 0;
	node[i].pJumpNode = (UDINT)&node[P_MENU];
	strcpy(node[i++].var.Format, "Return ");

	node[i].pHeadNode	= (UDINT)&node[P_PARAM_CONTIN_WELD];
	node[i].Type = N_SCROLL;
	strcpy(node[i++].var.Format, "*** Path Correction");

	node[i].pHeadNode	= (UDINT)&node[P_PARAM_CONTIN_WELD];
	node[i].Type = N_SCROLL + N_EDIT_IN_PLACE;
	node[i].var.Type = T_STRING;
	node[i].var.Var1ID = (h++);
	strcpy(node[i++].var.Format, "%s");

	node[i].pHeadNode	= (UDINT)&node[P_PARAM_CONTIN_WELD];
	node[i].Type = N_SCROLL + N_EDIT_IN_PLACE;
	node[i].var.Type = T_STRING;
	node[i].var.Var1ID = (h++);
	strcpy(node[i++].var.Format, "%s");

	node[i].pHeadNode	= (UDINT)&node[P_PARAM_CONTIN_WELD];
	node[i].Type = N_SCROLL;
	strcpy(node[i++].var.Format, "*** TVL in Contin. Weld");

	node[i].pHeadNode 	= (UDINT)&node[P_PARAM_CONTIN_WELD];
	node[i].Type = N_EDIT;
	node[i].MinUserLevel = 5;
	node[i].var.Type = T_SCALED;
	node[i].var.Var1ID = parCONTIN_TVL_RampDwn;
	strcpy(node[i++].var.Format, "%name%: %s");

	node[i].pHeadNode 	= (UDINT)&node[P_PARAM_CONTIN_WELD];
	node[i].Type = N_EDIT;
	node[i].MinUserLevel = 5;
	node[i].var.Type = T_SCALED;
	node[i].var.Var1ID = parCONTIN_TVL_RampUp;
	strcpy(node[i++].var.Format, "%name%: %s");

	node[i].pHeadNode	= (UDINT)&node[P_PARAM_CONTIN_WELD];
	node[i].Type = N_SCROLL;
	strcpy(node[i++].var.Format, "*** OSC Ramps");

	node[i].pHeadNode 	= (UDINT)&node[P_PARAM_CONTIN_WELD];
	node[i].Type = N_EDIT;
	node[i].MinUserLevel = 5;
	node[i].var.Type = T_SCALED;
	node[i].var.Var1ID = parOSC_RampDwn;
	strcpy(node[i++].var.Format, "%name%: %s");

	node[i].pHeadNode 	= (UDINT)&node[P_PARAM_CONTIN_WELD];
	node[i].Type = N_EDIT;
	node[i].MinUserLevel = 5;
	node[i].var.Type = T_SCALED;
	node[i].var.Var1ID = parOSC_RampUp;
	strcpy(node[i++].var.Format, "%name%: %s");

	node[i].pHeadNode	= (UDINT)&node[P_PARAM_CONTIN_WELD];
	node[i].Type = N_SCROLL;
	strcpy(node[i++].var.Format, "*** TIG AMP in Contin. Weld");

	node[i].pHeadNode 	= (UDINT)&node[P_PARAM_CONTIN_WELD];
	node[i].Type = N_EDIT;
	node[i].MinUserLevel = 5;
	node[i].var.Type = T_SCALED;
	node[i].var.Var1ID = parCONTIN_TIG_Percent;
	strcpy(node[i++].var.Format, "%name%: %s");

	node[i].pHeadNode 	= (UDINT)&node[P_PARAM_CONTIN_WELD];
	node[i].Type = N_EDIT;
	node[i].MinUserLevel = 5;
	node[i].var.Type = T_SCALED;
	node[i].var.Var1ID = parCONTIN_TIG_RampDwn;
	strcpy(node[i++].var.Format, "%name%: %s");

	/*
	node[i].pHeadNode 	= (UDINT)&node[P_PARAM_CONTIN_WELD];
	node[i].Type = N_EDIT;
	node[i].MinUserLevel = 5;
	node[i].var.Type = T_SCALED;
	node[i].var.Var1ID = parCONTIN_TIG_Dwell;
	strcpy(node[i++].var.Format, "%name%: %s");
	*/

	node[i].pHeadNode 	= (UDINT)&node[P_PARAM_CONTIN_WELD];
	node[i].Type = N_EDIT;
	node[i].MinUserLevel = 5;
	node[i].var.Type = T_SCALED;
	node[i].var.Var1ID = parCONTIN_TIG_RampUp;
	strcpy(node[i++].var.Format, "%name%: %s");

	node[i].pHeadNode	= (UDINT)&node[P_PARAM_CONTIN_WELD];
	node[i].Type = N_SCROLL;
	strcpy(node[i++].var.Format, "*** WF in Contin. Weld");

	node[i].pHeadNode 	= (UDINT)&node[P_PARAM_CONTIN_WELD];
	node[i].Type = N_EDIT;
	node[i].MinUserLevel = 5;
	node[i].var.Type = T_SCALED;
	node[i].var.Var1ID = parCONTIN_WF_RampDwn;
	strcpy(node[i++].var.Format, "%name%: %s");

	node[i].pHeadNode 	= (UDINT)&node[P_PARAM_CONTIN_WELD];
	node[i].Type = N_EDIT;
	node[i].MinUserLevel = 5;
	node[i].var.Type = T_SCALED;
	node[i].var.Var1ID = parCONTIN_WF_RampUp;
	strcpy(node[i++].var.Format, "%name%: %s");

	node[i].pHeadNode	= (UDINT)&node[P_PARAM_CONTIN_WELD];
	node[i].Type = N_SCROLL;
	strcpy(node[i++].var.Format, "*** WP in Contin. Weld");

	node[i].pHeadNode 	= (UDINT)&node[P_PARAM_CONTIN_WELD];
	node[i].Type = N_EDIT;
	node[i].MinUserLevel = 5;
	node[i].var.Type = T_SCALED;
	node[i].var.Var1ID = parCONTIN_WP_RampDwn;
	strcpy(node[i++].var.Format, "%name%: %s");

	node[i].pHeadNode 	= (UDINT)&node[P_PARAM_CONTIN_WELD];
	node[i].Type = N_EDIT;
	node[i].MinUserLevel = 5;
	node[i].var.Type = T_SCALED;
	node[i].var.Var1ID = parCONTIN_WP_RampUp;
	strcpy(node[i++].var.Format, "%name%: %s");

	/** P_PARAM_INDX **/
	i = P_PARAM_INDX;			h=varSTRING_HMI_0;
	SetPageDict(&cfg->PagesDict[n++] , P_PARAM_HW , "P_PARAM_INDX");

	node[i].pHeadNode	= (UDINT)&node[P_PARAM_INDX];
	node[i].Type = N_JUMP;
	node[i].JumpLineID = 0;
	node[i].pJumpNode = (UDINT)&node[P_PARAM];
	strcpy(node[i++].var.Format, "Return ");

	node[i].pHeadNode	= (UDINT)&node[P_PARAM_INDX];
	node[i].Type = N_EDIT;
	node[i].MinUserLevel = 5;
	node[i].var.Type = T_SCALED;
	node[i].var.Var1ID = parINDX_StepDist;
	//strcpy(node[i++].var.Format, "Step Dist. %s");
	strcpy(node[i++].var.Format, "%name%: %s");

	node[i].pHeadNode	= (UDINT)&node[P_PARAM_INDX];
	node[i].Type = N_EDIT;
	node[i].MinUserLevel = 5;
	node[i].var.Type = T_SCALED;
	node[i].var.Var1ID = parINDX_StepAfterBeats;
	//strcpy(node[i++].var.Format, "Step After Beats %s");
	strcpy(node[i++].var.Format, "%name%: %s");

	node[i].pHeadNode	= (UDINT)&node[P_PARAM_INDX];
	node[i].Type = N_EDIT;
	node[i].MinUserLevel = 5;
	node[i].var.Type = T_SCALED;
	node[i].var.Var1ID = parINDX_StepVel;
	//strcpy(node[i++].var.Format, "Step Vel. %s");
	strcpy(node[i++].var.Format, "%name%: %s");

	node[i].pHeadNode	= (UDINT)&node[P_PARAM_INDX];
	node[i].Type = N_EDIT;
	node[i].MinUserLevel = 5;
	node[i].var.Type = T_SCALED;
	node[i].var.Var1ID = parINDX_JogSpeedDirCntrl;
	//strcpy(node[i++].var.Format, "Jog Speed %s");
	strcpy(node[i++].var.Format, "%name%: %s");

	/*
	node[i].pHeadNode	= (UDINT)&node[P_PARAM_INDX];
	node[i].Type = N_SCROLL;
	strcpy(node[i++].var.Format, "JOG ONLY A");

	node[i].pHeadNode	= (UDINT)&node[P_PARAM_INDX];
	node[i].Type = N_SCROLL;
	strcpy(node[i++].var.Format, "JOG ONLY B");

	node[i].pHeadNode	= (UDINT)&node[P_PARAM_INDX];
	node[i].Type = N_SCROLL +  N_EVENT ;
	node[i].Event = EVNT_SET_INDX_ZERO;
	strcpy(node[i++].var.Format, "Set Zero");
*/

	/** P_PARAM_GAS **/
	i = P_PARAM_GAS;			h=varSTRING_HMI_0;
	SetPageDict(&cfg->PagesDict[n++] , P_PARAM_GAS , "P_PARAM_GAS");

	node[i].pHeadNode	= (UDINT)&node[P_PARAM_GAS];
	node[i].Type = N_JUMP;
	node[i].JumpLineID = 0;
	node[i].pJumpNode = (UDINT)&node[P_PARAM];
	strcpy(node[i++].var.Format, "Return ");

	node[i].pHeadNode	= (UDINT)&node[P_PARAM_GAS];
	node[i].Type = N_EDIT;
	node[i].MinUserLevel = 5;
	node[i].var.Type = T_SCALED;
	node[i].var.Var1ID = parGAS_PrePurgeTm;
	//strcpy(node[i++].var.Format, "PREPURGE %s");
	strcpy(node[i++].var.Format, "%name%: %s");

	node[i].pHeadNode 	= (UDINT)&node[P_PARAM_GAS];
	node[i].Type = N_SCROLL + N_NO_PREFIX;
	node[i].MinUserLevel = 5;
	strcpy(node[i++].var.Format, "******* MSC. *******");

	node[i].pHeadNode	= (UDINT)&node[P_PARAM_GAS];
	node[i].Type = N_EDIT;
	node[i].MinUserLevel = 5;
	node[i].var.Type = T_SCALED;
	node[i].var.Var1ID = parGAS_Tmo;
	//strcpy(node[i++].var.Format, "Argon TMO: %s");
	strcpy(node[i++].var.Format, "%name%: %s");

	node[i].pHeadNode	= (UDINT)&node[P_PARAM_GAS];
	node[i].Type = N_EDIT;
	node[i].MinUserLevel = 5;
	node[i].var.Type = T_SCALED;
	node[i].var.Var1ID = parCOOL_Tmo;
	//strcpy(node[i++].var.Format, "Cool TMO: %s");
	strcpy(node[i++].var.Format, "%name%: %s");

	node[i].pHeadNode	= (UDINT)&node[P_PARAM_GAS];
	node[i].Type = N_SCROLL + N_NO_PREFIX;
	node[i].MinUserLevel = 5;
	strcpy(node[i++].var.Format, "**** CALCULATED ****");

	node[i].pHeadNode	= (UDINT)&node[P_PARAM_GAS];
	node[i].Type = N_EDIT;
	node[i].MinUserLevel = 5;
	node[i].var.Type = T_SCALED;
	node[i].var.Var1ID = parGAS_PostPurgeTm;
	//strcpy(node[i++].var.Format, "PostPurge %s");
	strcpy(node[i++].var.Format, "%name%: %s");

	/** P_VAR_SETUP **/
	i = P_VAR_SETUP;			h=varSTRING_HMI_0;
	SetPageDict(&cfg->PagesDict[n++] , P_VAR_SETUP , "P_VAR_SETUP");

	node[i].pHeadNode	= (UDINT)&node[P_VAR_SETUP];
	node[i].Type = N_JUMP;
	node[i].JumpLineID = 0;
	node[i].pJumpNode = (UDINT)&node[P_MENU];
	strcpy(node[i++].var.Format, "Return ");

	node[i].pHeadNode	= (UDINT)&node[P_VAR_SETUP];
	node[i].Type = N_EDIT;
	node[i].var.Type = T_SCALED;
	node[i].var.Var1ID = parGEN_AmpRead;
	//strcpy(node[i++].var.Format, "Cal.Amp: %s");
	strcpy(node[i++].var.Format, "%name%: %s");

	node[i].pHeadNode	= (UDINT)&node[P_VAR_SETUP];
	node[i].Type = N_EDIT;
	node[i].var.Type = T_SCALED;
	node[i].var.Var1ID = parGEN_CalibDist;
	//strcpy(node[i++].var.Format, "Cal.Dist: %s");
	strcpy(node[i++].var.Format, "%name%: %s");

	node[i].pHeadNode	= (UDINT)&node[P_VAR_SETUP];
	node[i].Type = N_EDIT;
	node[i].var.Type = T_SCALED;
	node[i].var.Var1ID = parGEN_CalibDist_2;
	//strcpy(node[i++].var.Format, "Cal.Dist: %s");
	strcpy(node[i++].var.Format, "%name%: %s");

	node[i].pHeadNode	= (UDINT)&node[P_VAR_SETUP];
	node[i].Type = N_EDIT;
	node[i].var.Type = T_SCALED;
	node[i].var.Var1ID = parGEN_CalibTime;
	//strcpy(node[i++].var.Format, "Cal.Time: %s");
	strcpy(node[i++].var.Format, "%name%: %s");

	node[i].pHeadNode	= (UDINT)&node[P_VAR_SETUP];
	node[i].Type = N_EDIT;
	node[i].var.Type = T_SCALED;
	node[i].var.Var1ID = varOSC_Centr;
	//strcpy(node[i++].var.Format, "actOSC Centr: %s");
	strcpy(node[i++].var.Format, "%name%: %s");

	node[i].pHeadNode	= (UDINT)&node[P_VAR_SETUP];
	node[i].Type = N_EDIT;
	node[i].var.Type = T_SCALED;
	node[i].var.Var1ID = varOSC_CurPos;
	//strcpy(node[i++].var.Format, "actOSC Pos: %s");
	strcpy(node[i++].var.Format, "%name%: %s");

	node[i].pHeadNode	= (UDINT)&node[P_VAR_SETUP];
	node[i].Type = N_EDIT;
	node[i].var.Type = T_SCALED;
	node[i].var.Var1ID = varHW_Amp_Cmd;
	//strcpy(node[i++].var.Format, "actHW Amp: %s");
	strcpy(node[i++].var.Format, "%name%: %s");

	node[i].pHeadNode	= (UDINT)&node[P_VAR_SETUP];
	node[i].Type = N_EDIT;
	node[i].var.Type = T_SCALED;
	node[i].var.Var1ID = varCurArc_Volt;
	//strcpy(node[i++].var.Format, "actTIG Volt: %s");
	strcpy(node[i++].var.Format, "%name%: %s");

	node[i].pHeadNode	= (UDINT)&node[P_VAR_SETUP];
	node[i].Type = N_EDIT;
	node[i].var.Type = T_SCALED;
	node[i].var.Var1ID = varCurTIG_Amp;
	//strcpy(node[i++].var.Format, "actTIG Amp: %s");
	strcpy(node[i++].var.Format, "%name%: %s");

	node[i].pHeadNode	= (UDINT)&node[P_VAR_SETUP];
	node[i].Type = N_EDIT;
	node[i].var.Type = T_SCALED;
	node[i].var.Var1ID = varTIG_Amp_Cmd;
	//strcpy(node[i++].var.Format, "cmdTIG Amp: %s");
	strcpy(node[i++].var.Format, "%name%: %s");

	node[i].pHeadNode	= (UDINT)&node[P_VAR_SETUP];
	node[i].Type = N_EDIT;
	node[i].var.Type = T_SCALED;
	node[i].var.Var1ID = varCurTVL_Vel;
	//strcpy(node[i++].var.Format, "actTVL Vel: %s");
	strcpy(node[i++].var.Format, "%name%: %s");

	node[i].pHeadNode	= (UDINT)&node[P_VAR_SETUP];
	node[i].Type = N_EDIT;
	node[i].var.Type = T_SCALED;
	node[i].var.Var1ID = varCurWF_Vel;
	//strcpy(node[i++].var.Format, "actWF Vel: %s");
	strcpy(node[i++].var.Format, "%name%: %s");

	node[i].pHeadNode	= (UDINT)&node[P_VAR_SETUP];
	node[i].Type = N_EDIT;
	node[i].var.Type = T_SCALED;
	node[i].var.Var1ID = varCurWP_Vel;
	//strcpy(node[i++].var.Format, "actWP Freq: %s");
	strcpy(node[i++].var.Format, "%name%: %s");

	node[i].pHeadNode	= (UDINT)&node[P_VAR_SETUP];
	node[i].Type = N_EDIT;
	node[i].var.Type = T_SCALED;
	node[i].var.Var1ID = varCurWFDist;
	//strcpy(node[i++].var.Format, "actWF Dist: %s");
	strcpy(node[i++].var.Format, "%name%: %s");

	/** P_PARAM_GLOBAL **/
	i = P_PARAM_GLOBAL;			h=varSTRING_HMI_0;
	SetPageDict(&cfg->PagesDict[n++] , P_PARAM_GLOBAL , "P_PARAM_GLOBAL");

	node[i].pHeadNode	= (UDINT)&node[P_PARAM_GLOBAL];
	node[i].Type = N_SCROLL + N_EDIT_IN_PLACE;
	node[i].var.Type = T_STRING;
	node[i].var.Var1ID = (h++);
	strcpy(node[i++].var.Format, "%s");

	node[i].pHeadNode	= (UDINT)&node[P_PARAM_GLOBAL];
	node[i].Type = N_SCROLL + N_EDIT_IN_PLACE;
	node[i].var.Type = T_STRING;
	node[i].var.Var1ID = (h++);
	strcpy(node[i++].var.Format, "%s");

	node[i].pHeadNode	= (UDINT)&node[P_PARAM_GLOBAL];
	node[i].Type = N_SCROLL  + N_EDIT_IN_PLACE;
	node[i].var.Type = T_STRING;
	node[i].var.Var1ID = (h++);
	strcpy(node[i++].var.Format, "%s");

	// Use Mapping
	node[i].pHeadNode	= (UDINT)&node[P_PARAM_GLOBAL];
	node[i].Type = N_SCROLL  + N_EDIT_IN_PLACE;
	node[i].var.Type = T_STRING;
	node[i].var.Var1ID = (h++);
	strcpy(node[i++].var.Format, "%s");

	/// Auto Start
	node[i].pHeadNode	= (UDINT)&node[P_PARAM_GLOBAL];
	node[i].Type = N_SCROLL  + N_EDIT_IN_PLACE;
	node[i].var.Type = T_STRING;
	node[i].var.Var1ID = (h++);
	strcpy(node[i++].var.Format, "%s");

	// Auto Start Time
	node[i].pHeadNode	= (UDINT)&node[P_PARAM_GLOBAL];
	node[i].Type = N_SCROLL  + N_EDIT_IN_PLACE;
	node[i].var.Type = T_STRING;
	node[i].var.Var1ID = (h++);
	strcpy(node[i++].var.Format, "%s");

	// Single Start Sound ON / OFF
	node[i].pHeadNode	= (UDINT)&node[P_PARAM_GLOBAL];
	node[i].Type = N_SCROLL  + N_EDIT_IN_PLACE;
	node[i].var.Type = T_STRING;
	node[i].var.Var1ID = (h++);
	strcpy(node[i++].var.Format, "%s");

	// Start Sound Time
	node[i].pHeadNode	= (UDINT)&node[P_PARAM_GLOBAL];
	node[i].Type = N_SCROLL  + N_EDIT_IN_PLACE;
	node[i].var.Type = T_STRING;
	node[i].var.Var1ID = (h++);
	strcpy(node[i++].var.Format, "%s");

	// INDEX Enable
	node[i].pHeadNode	= (UDINT)&node[P_PARAM_GLOBAL];
	node[i].Type = N_SCROLL  + N_EDIT_IN_PLACE;
	node[i].var.Type = T_STRING;
	node[i].var.Var1ID = (h++);
	strcpy(node[i++].var.Format, "%s");

	// INDEX Direction
	node[i].pHeadNode	= (UDINT)&node[P_PARAM_GLOBAL];
	node[i].Type = N_SCROLL  + N_EDIT_IN_PLACE;
	node[i].var.Type = T_STRING;
	node[i].var.Var1ID = (h++);
	strcpy(node[i++].var.Format, "%s");

	//SETUP_ZONE_CENTR
	node[i].pHeadNode	= (UDINT)&node[P_PARAM_GLOBAL];
	node[i].Type = N_SCROLL  + N_EDIT_IN_PLACE;
	node[i].var.Type = T_STRING;
	node[i].var.Var1ID = (h++);
	strcpy(node[i++].var.Format, "%s");

	// SETUP_TWO_TORCH
	node[i].pHeadNode	= (UDINT)&node[P_PARAM_GLOBAL];
	node[i].Type = N_SCROLL  + N_EDIT_IN_PLACE;
	node[i].var.Type = T_STRING;
	node[i].var.Var1ID = (h++);
	strcpy(node[i++].var.Format, "%s");

	// SETUP_ONE_UP
	node[i].pHeadNode	= (UDINT)&node[P_PARAM_GLOBAL];
	node[i].Type = N_SCROLL  + N_EDIT_IN_PLACE;
	node[i].var.Type = T_STRING;
	node[i].var.Var1ID = (h++);
	strcpy(node[i++].var.Format, "%s");

	//SETUP_CONTIN_WELD
	node[i].pHeadNode	= (UDINT)&node[P_PARAM_GLOBAL];
	node[i].Type = N_SCROLL  + N_EDIT_IN_PLACE;
	node[i].var.Type = T_STRING;
	node[i].var.Var1ID = (h++);
	strcpy(node[i++].var.Format, "%s");

	//SETUP_TVL_ENC_SET
	node[i].pHeadNode	= (UDINT)&node[P_PARAM_GLOBAL];
	node[i].Type = N_SCROLL  + N_EDIT_IN_PLACE;
	node[i].var.Type = T_STRING;
	node[i].var.Var1ID = (h++);
	strcpy(node[i++].var.Format, "%s");

	// SETUP_TVL_SEC_ENC
	node[i].pHeadNode	= (UDINT)&node[P_PARAM_GLOBAL];
	node[i].Type = N_SCROLL  + N_EDIT_IN_PLACE;
	node[i].var.Type = T_STRING;
	node[i].var.Var1ID = (h++);
	strcpy(node[i++].var.Format, "%s");

	node[i].pHeadNode	= (UDINT)&node[P_PARAM_GLOBAL];
	node[i].Type = N_SCROLL;
	strcpy(node[i++].var.Format, " ******** ");

	/// HEAD TYPE

	node[i].pHeadNode	= (UDINT)&node[P_PARAM_GLOBAL];
	node[i].Type = N_SCROLL  + N_EDIT_IN_PLACE;
	node[i].var.Type = T_STRING;
	node[i].var.Var1ID = (h++);
	strcpy(node[i++].var.Format, "%s");

	/// Legacy AVC

	node[i].pHeadNode	= (UDINT)&node[P_PARAM_GLOBAL];
	node[i].Type = N_SCROLL  + N_EDIT_IN_PLACE;
	node[i].var.Type = T_STRING;
	node[i].var.Var1ID = (h++);
	strcpy(node[i++].var.Format, "%s");

	/// WF Swap
	node[i].pHeadNode	= (UDINT)&node[P_PARAM_GLOBAL];
	node[i].Type = N_SCROLL  + N_EDIT_IN_PLACE;
	node[i].var.Type = T_STRING;
	node[i].var.Var1ID = (h++);
	strcpy(node[i++].var.Format, "%s");

	/// WF Stop Ramp
	node[i].pHeadNode	= (UDINT)&node[P_PARAM_GLOBAL];
	node[i].Type = N_SCROLL  + N_EDIT_IN_PLACE;
	node[i].var.Type = T_STRING;
	node[i].var.Var1ID = (h++);
	strcpy(node[i++].var.Format, "%s");

	/// WF Start Ramp
	h=varSTRING_HMI_0;
	node[i].pHeadNode	= (UDINT)&node[P_PARAM_GLOBAL];
	node[i].Type = N_SCROLL  + N_EDIT_IN_PLACE;
	node[i].var.Type = T_STRING;
	node[i].var.Var1ID = (h++);
	strcpy(node[i++].var.Format, "%s");

	// P_MODE_WF_CALIB_PAR
	i= P_MODE_WF_CALIB_PAR;			h=varSTRING_HMI_0;
	SetPageDict(&cfg->PagesDict[n++] , P_MODE_WF_CALIB_PAR , "P_MODE_WF_CALIB_PAR");

	node[i].pHeadNode	= (UDINT)&node[P_MODE_WF_CALIB_PAR];
	node[i].Type = N_SCROLL + N_EVENT ;
	node[i].Event = EVNT_OK;
	node[i].var.Type = T_STRING;
	node[i].var.Var1ID = (h++);
	strcpy(node[i++].var.Format, "%s");

	node[i].pHeadNode	= (UDINT)&node[P_MODE_WF_CALIB_PAR];
	node[i].Type = N_EDIT;
	node[i].var.Type = T_SCALED;
	node[i].var.Var1ID = parWF_CalibVel1;
	//strcpy(node[i++].var.Format, "Low Vel: %s");
	strcpy(node[i++].var.Format, "%name%: %s");

	node[i].pHeadNode	= (UDINT)&node[P_MODE_WF_CALIB_PAR];
	node[i].Type = N_EDIT;
	node[i].var.Type = T_SCALED;
	node[i].var.Var1ID = parWF_CalibVel2;
	//strcpy(node[i++].var.Format, "High Vel: %s");
	strcpy(node[i++].var.Format, "%name%: %s");

	node[i].pHeadNode	= (UDINT)&node[P_MODE_WF_CALIB_PAR];
	node[i].Type = N_EDIT;
	node[i].var.Type = T_SCALED;
	node[i].var.Var1ID = parGEN_CalibDist;
	//strcpy(node[i++].var.Format, "Length: %s");
	strcpy(node[i++].var.Format, "%name%: %s");

	node[i].pHeadNode	= (UDINT)&node[P_MODE_WF_CALIB_PAR];
	node[i].Type = N_EDIT;
	node[i].var.Type = T_SCALED;
	node[i].var.Var1ID = parGEN_CalibDist_2;
	//strcpy(node[i++].var.Format, "Length: %s");
	strcpy(node[i++].var.Format, "%name%: %s");

	node[i].pHeadNode	= (UDINT)&node[P_MODE_WF_CALIB_PAR];
	node[i].Type = N_SCROLL;
	node[i].var.Type = T_STRING;
	node[i].var.Var1ID = (h++);
	strcpy(node[i++].var.Format, "%s");

	node[i].pHeadNode	= (UDINT)&node[P_MODE_WF_CALIB_PAR];
	node[i].Type = N_SCROLL + N_EVENT ;
	node[i].Event = EVNT_CANCEL;
	node[i].var.Type = T_STRING;
	node[i].var.Var1ID = (h++);
	strcpy(node[i++].var.Format, "%s");

	// P_MODE_WF_CALIB
	i= P_MODE_WF_CALIB;			h=varSTRING_HMI_0;
	SetPageDict(&cfg->PagesDict[n++] , P_MODE_WF_CALIB , "P_MODE_WF_CALIB");

	node[i].pHeadNode	= (UDINT)&node[P_MODE_WF_CALIB];
	node[i].Type = N_SCROLL +  N_EVENT ;
	node[i].Event = EVNT_CANCEL;
	node[i].var.Type = T_STRING;
	node[i].var.Var1ID = (h++);
	strcpy(node[i++].var.Format, "%s");

	node[i].pHeadNode	= (UDINT)&node[P_MODE_WF_CALIB];
	node[i].Type = N_EDIT;
	node[i].var.Type = T_SCALED;
	node[i].var.Var1ID = parGEN_CalibDist1;
	//strcpy(node[i++].var.Format, "(1)Length at Head A Low Vel.:  %s");
	strcpy(node[i++].var.Format, "%name%: %s");

	node[i].pHeadNode	= (UDINT)&node[P_MODE_WF_CALIB];
	node[i].Type = N_EDIT;
	node[i].var.Type = T_SCALED;
	node[i].var.Var1ID = parGEN_CalibDist2;
	//strcpy(node[i++].var.Format, "(2)Length at Head A High Vel.:  %s");
	strcpy(node[i++].var.Format, "%name%: %s");

	node[i].pHeadNode	= (UDINT)&node[P_MODE_WF_CALIB];
	node[i].Type = N_EDIT;
	node[i].var.Type = T_SCALED;
	node[i].var.Var1ID = parGEN_CalibDist3;
	//strcpy(node[i++].var.Format, "(3)Length at Head B Low Vel.:  %s");
	strcpy(node[i++].var.Format, "%name%: %s");

	node[i].pHeadNode	= (UDINT)&node[P_MODE_WF_CALIB];
	node[i].Type = N_EDIT;
	node[i].var.Type = T_SCALED;
	node[i].var.Var1ID = parGEN_CalibDist4;
	//strcpy(node[i++].var.Format, "(4)Length at Head B High Vel.:  %s");
	strcpy(node[i++].var.Format, "%name%: %s");

	node[i].pHeadNode	= (UDINT)&node[P_MODE_WF_CALIB];
	node[i].Type = N_SCROLL +  N_EVENT ;
	node[i].Event = EVNT_OK;
	node[i].var.Type = T_STRING;
	node[i].var.Var1ID = (h++);
	strcpy(node[i++].var.Format, " %s");

	// P_MODE_WF_CALIB_VER
	i= P_MODE_WF_CALIB_VER;			h=varSTRING_HMI_0;
	SetPageDict(&cfg->PagesDict[n++] , P_MODE_WF_CALIB_VER , "P_MODE_WF_CALIB_VER");

	node[i].pHeadNode	= (UDINT)&node[P_MODE_WF_CALIB_VER];
	node[i].Type = N_SCROLL +  N_EVENT ;
	node[i].Event = EVNT_CANCEL;
	strcpy(node[i++].var.Format, "Repeat !!!");

	node[i].pHeadNode	= (UDINT)&node[P_MODE_WF_CALIB_VER];
	node[i].Type = N_SCROLL;
	node[i].var.Type = T_STRING;
	node[i].var.Var1ID = (h++);
	strcpy(node[i++].var.Format, "%s");

	node[i].pHeadNode	= (UDINT)&node[P_MODE_WF_CALIB_VER];
	node[i].Type = N_SCROLL;
	node[i].var.Type = T_STRING;
	node[i].var.Var1ID = (h++);
	strcpy(node[i++].var.Format, "%s");

	node[i].pHeadNode	= (UDINT)&node[P_MODE_WF_CALIB_VER];
	node[i].Type = N_SCROLL;
	node[i].var.Type = T_STRING;
	node[i].var.Var1ID = (h++);
	strcpy(node[i++].var.Format, "%s");

	node[i].pHeadNode	= (UDINT)&node[P_MODE_WF_CALIB_VER];
	node[i].Type = N_SCROLL +  N_EVENT ;
	node[i].Event = EVNT_OK;
	strcpy(node[i++].var.Format, "Save Calibration !!!");

	//P_MODE_TIG_PS_CALIB_PAR
	i= P_MODE_TIG_PS_CALIB_PAR;			h=varSTRING_HMI_0;
	SetPageDict(&cfg->PagesDict[n++] , P_MODE_TIG_PS_CALIB_PAR , "P_MODE_TIG_PS_CALIB_PAR");

	node[i].pHeadNode	= (UDINT)&node[P_MODE_TIG_PS_CALIB_PAR];
	node[i].Type = N_SCROLL + N_EVENT ;
	node[i].Event = EVNT_OK;
	node[i].var.Type = T_STRING;
	node[i].var.Var1ID = (h++);
	strcpy(node[i++].var.Format, "%s");

	node[i].pHeadNode	= (UDINT)&node[P_MODE_TIG_PS_CALIB_PAR];
	node[i].Type = N_EDIT;
	node[i].var.Type = T_SCALED;
	node[i].var.Var1ID = parTIG_CalibAmp1;
	//strcpy(node[i++].var.Format, "Low Amp: %s");
	strcpy(node[i++].var.Format, "%name%: %s");

	node[i].pHeadNode	= (UDINT)&node[P_MODE_TIG_PS_CALIB_PAR];
	node[i].Type = N_EDIT;
	node[i].var.Type = T_SCALED;
	node[i].var.Var1ID = parTIG_CalibAmp2;
	//strcpy(node[i++].var.Format, "High Amp: %s");
	strcpy(node[i++].var.Format, "%name%: %s");

	node[i].pHeadNode	= (UDINT)&node[P_MODE_TIG_PS_CALIB_PAR];
	node[i].Type = N_EDIT;
	node[i].var.Type = T_ENUM;
	node[i].var.Var1ID = parENUM_TIG_Cal_Mode;
	strcpy(node[i++].var.Format, "%name%: %s");

	node[i].pHeadNode	= (UDINT)&node[P_MODE_TIG_PS_CALIB_PAR];
	node[i].Type = N_SCROLL;
	node[i].var.Type = T_STRING;
	node[i].var.Var1ID = (h++);
	strcpy(node[i++].var.Format, "%s");

	node[i].pHeadNode	= (UDINT)&node[P_MODE_TIG_PS_CALIB_PAR];
	node[i].Type = N_SCROLL + N_EVENT;
	node[i].Event = EVNT_CANCEL;
	node[i].var.Type = T_STRING;
	node[i].var.Var1ID = (h++);
	strcpy(node[i++].var.Format, "%s");

	//P_MODE_TIG_PS_CALIB
	i= P_MODE_TIG_PS_CALIB;			h=varSTRING_HMI_0;
	SetPageDict(&cfg->PagesDict[n++] , P_MODE_TIG_PS_CALIB , "P_MODE_TIG_PS_CALIB");

	node[i].pHeadNode	= (UDINT)&node[P_MODE_TIG_PS_CALIB];
	node[i].Type = N_SCROLL +  N_EVENT ;
	node[i].Event = EVNT_CANCEL;
	node[i].var.Type = T_STRING;
	node[i].var.Var1ID = (h++);
	strcpy(node[i++].var.Format, "%s");

	node[i].pHeadNode	= (UDINT)&node[P_MODE_TIG_PS_CALIB];
	node[i].Type = N_EDIT;
	node[i].var.Type = T_SCALED;
	node[i].var.Var1ID = parGEN_CalibAmp1;
	//strcpy(node[i++].var.Format, "(1)Low Amps:  %s");
	strcpy(node[i++].var.Format, "%name%: %s");

	node[i].pHeadNode	= (UDINT)&node[P_MODE_TIG_PS_CALIB];
	node[i].Type = N_EDIT;
	node[i].var.Type = T_SCALED;
	node[i].var.Var1ID = parGEN_CalibAmp2;
	//strcpy(node[i++].var.Format, "(2)High Amps: %s");
	strcpy(node[i++].var.Format, "%name%: %s");

	node[i].pHeadNode	= (UDINT)&node[P_MODE_TIG_PS_CALIB];
	node[i].Type = N_SCROLL +  N_EVENT ;
	node[i].Event = EVNT_OK;
	node[i].var.Type = T_STRING;
	node[i].var.Var1ID = (h++);
	strcpy(node[i++].var.Format, " %s");

	// P_MODE_TIG_PS_CALIB_VER
	i= P_MODE_TIG_PS_CALIB_VER;			h=varSTRING_HMI_0;
	SetPageDict(&cfg->PagesDict[n++] , P_MODE_TIG_PS_CALIB_VER , "P_MODE_TIG_PS_CALIB_VER");

	node[i].pHeadNode	= (UDINT)&node[P_MODE_TIG_PS_CALIB_VER];
	node[i].Type = N_SCROLL +  N_EVENT ;
	node[i].Event = EVNT_CANCEL;
	strcpy(node[i++].var.Format, "Repeat !!!");

	node[i].pHeadNode	= (UDINT)&node[P_MODE_TIG_PS_CALIB_VER];
	node[i].Type = N_SCROLL;
	node[i].var.Type = T_STRING;
	node[i].var.Var1ID = (h++);
	strcpy(node[i++].var.Format, "%s");

	node[i].pHeadNode	= (UDINT)&node[P_MODE_TIG_PS_CALIB_VER];
	node[i].Type = N_SCROLL;
	node[i].var.Type = T_STRING;
	node[i].var.Var1ID = (h++);
	strcpy(node[i++].var.Format, "%s");

	node[i].pHeadNode	= (UDINT)&node[P_MODE_TIG_PS_CALIB_VER];
	node[i].Type = N_SCROLL +  N_EVENT ;
	node[i].Event = EVNT_OK;
	strcpy(node[i++].var.Format, "Save Calibration !!!");

	//P_MODE_HW_PS_CALIB_PAR
	i= P_MODE_HW_PS_CALIB_PAR;			h=varSTRING_HMI_0;
	SetPageDict(&cfg->PagesDict[n++] , P_MODE_HW_PS_CALIB_PAR , "P_MODE_HW_PS_CALIB_PAR");

	node[i].pHeadNode	= (UDINT)&node[P_MODE_HW_PS_CALIB_PAR];
	node[i].Type = N_SCROLL + N_EVENT ;
	node[i].Event = EVNT_OK;
	node[i].var.Type = T_STRING;
	node[i].var.Var1ID = (h++);
	strcpy(node[i++].var.Format, "%s");

	node[i].pHeadNode	= (UDINT)&node[P_MODE_HW_PS_CALIB_PAR];
	node[i].Type = N_EDIT;
	node[i].var.Type = T_SCALED;
	node[i].var.Var1ID = parHW_CalibAmp1;
	//strcpy(node[i++].var.Format, "Low Amp: %s");
	strcpy(node[i++].var.Format, "%name%: %s");

	node[i].pHeadNode	= (UDINT)&node[P_MODE_HW_PS_CALIB_PAR];
	node[i].Type = N_EDIT;
	node[i].var.Type = T_SCALED;
	node[i].var.Var1ID = parHW_CalibAmp2;
	//strcpy(node[i++].var.Format, "High Amp: %s");
	strcpy(node[i++].var.Format, "%name%: %s");

	node[i].pHeadNode	= (UDINT)&node[P_MODE_HW_PS_CALIB_PAR];
	node[i].Type = N_SCROLL;
	node[i].var.Type = T_STRING;
	node[i].var.Var1ID = (h++);
	strcpy(node[i++].var.Format, "%s");

	node[i].pHeadNode	= (UDINT)&node[P_MODE_HW_PS_CALIB_PAR];
	node[i].Type = N_SCROLL + N_EVENT;
	node[i].Event = EVNT_CANCEL;
	node[i].var.Type = T_STRING;
	node[i].var.Var1ID = (h++);
	strcpy(node[i++].var.Format, "%s");

	//P_MODE_HW_PS_CALIB
	i= P_MODE_HW_PS_CALIB;			h=varSTRING_HMI_0;
	SetPageDict(&cfg->PagesDict[n++] , P_MODE_HW_PS_CALIB , "P_MODE_HW_PS_CALIB");

	node[i].pHeadNode	= (UDINT)&node[P_MODE_HW_PS_CALIB];
	node[i].Type = N_SCROLL +  N_EVENT ;
	node[i].Event = EVNT_CANCEL;
	node[i].var.Type = T_STRING;
	node[i].var.Var1ID = (h++);
	strcpy(node[i++].var.Format, "%s");

	node[i].pHeadNode	= (UDINT)&node[P_MODE_HW_PS_CALIB];
	node[i].Type = N_EDIT;
	node[i].var.Type = T_SCALED;
	node[i].var.Var1ID = parGEN_CalibAmp1;
	//strcpy(node[i++].var.Format, "(1)Low Amps:  %s");
	strcpy(node[i++].var.Format, "%name%: %s");

	node[i].pHeadNode	= (UDINT)&node[P_MODE_HW_PS_CALIB];
	node[i].Type = N_EDIT;
	node[i].var.Type = T_SCALED;
	node[i].var.Var1ID = parGEN_CalibAmp2;
	//strcpy(node[i++].var.Format, "(2)High Amps: %s");
	strcpy(node[i++].var.Format, "%name%: %s");

	node[i].pHeadNode	= (UDINT)&node[P_MODE_HW_PS_CALIB];
	node[i].Type = N_SCROLL +  N_EVENT ;
	node[i].Event = EVNT_OK;
	node[i].var.Type = T_STRING;
	node[i].var.Var1ID = (h++);
	strcpy(node[i++].var.Format, " %s");

	// P_MODE_HW_PS_CALIB_PAR
	i= P_MODE_HW_PS_CALIB_VER;			h=varSTRING_HMI_0;
	SetPageDict(&cfg->PagesDict[n++] , P_MODE_HW_PS_CALIB_VER , "P_MODE_HW_PS_CALIB_VER");

	node[i].pHeadNode	= (UDINT)&node[P_MODE_HW_PS_CALIB_VER];
	node[i].Type = N_SCROLL +  N_EVENT ;
	node[i].Event = EVNT_CANCEL;
	strcpy(node[i++].var.Format, "Repeat !!!");

	node[i].pHeadNode	= (UDINT)&node[P_MODE_HW_PS_CALIB_VER];
	node[i].Type = N_SCROLL;
	node[i].var.Type = T_STRING;
	node[i].var.Var1ID = (h++);
	strcpy(node[i++].var.Format, "%s");

	node[i].pHeadNode	= (UDINT)&node[P_MODE_HW_PS_CALIB_VER];
	node[i].Type = N_SCROLL;
	node[i].var.Type = T_STRING;
	node[i].var.Var1ID = (h++);
	strcpy(node[i++].var.Format, "%s");

	node[i].pHeadNode	= (UDINT)&node[P_MODE_HW_PS_CALIB_VER];
	node[i].Type = N_SCROLL +  N_EVENT ;
	node[i].Event = EVNT_OK;
	strcpy(node[i++].var.Format, "Save Calibration !!!");

	// P_MODE_OSC_LIMIT_CALIB
	i= P_MODE_OSC_LIMIT_CALIB;			h=varSTRING_HMI_0;
	SetPageDict(&cfg->PagesDict[n++] , P_MODE_OSC_LIMIT_CALIB , "P_MODE_OSC_LIMIT_CALIB");

	node[i].pHeadNode	= (UDINT)&node[P_MODE_OSC_LIMIT_CALIB];
	node[i].Type = N_SCROLL +  N_EVENT ;
	node[i].Event = EVNT_SWAP_HEAD;
	node[i].var.Type = T_STRING;
	node[i].var.Var1ID = (h++);
	strcpy(node[i++].var.Format, "%s");

	node[i].pHeadNode	= (UDINT)&node[P_MODE_OSC_LIMIT_CALIB];
	node[i].Type = N_SCROLL;
	node[i].var.Type = T_SCALED;
	node[i].var.Var1ID = varOSC_CurRawPos;
	//strcpy(node[i++].var.Format, "actPos FBK: %s");
	strcpy(node[i++].var.Format, "%name%: %s");

	node[i].pHeadNode	= (UDINT)&node[P_MODE_OSC_LIMIT_CALIB];
	node[i].Type = N_SCROLL +  N_EVENT ;
	node[i].Event = EVNT_OSC_POS_LIMIT_SET;
	strcpy(node[i++].var.Format, "Store Pos Limit");

	node[i].pHeadNode	= (UDINT)&node[P_MODE_OSC_LIMIT_CALIB];
	node[i].Type = N_SCROLL +  N_EVENT ;
	node[i].Event = EVNT_OSC_NEG_LIMIT_SET;
	strcpy(node[i++].var.Format, "Store Neg Limit");

	// P_MODE_TIG_FBK_CALIB
	i= P_MODE_TIG_FBK_CALIB;			h=varSTRING_HMI_0;
	SetPageDict(&cfg->PagesDict[n++] , P_MODE_TIG_FBK_CALIB , "P_MODE_TIG_FBK_CALIB");

	node[i].pHeadNode	= (UDINT)&node[P_MODE_TIG_FBK_CALIB];
	node[i].Type = N_SCROLL;
	node[i].var.Type = T_SCALED;
	node[i].var.Var1ID = varCurArc_Volt;
	//strcpy(node[i++].var.Format, "act Arc: %s");
	strcpy(node[i++].var.Format, "%name%: %s");

	node[i].pHeadNode	= (UDINT)&node[P_MODE_TIG_FBK_CALIB];
	node[i].Type = N_SCROLL +   N_EDIT_IN_PLACE ;
	node[i].var.Type = T_STRING;
	node[i].var.Var1ID = (h++);
	strcpy(node[i++].var.Format, "%s");

	node[i].pHeadNode	= (UDINT)&node[P_MODE_TIG_FBK_CALIB];
	node[i].Type = N_SCROLL +  N_EVENT ;
	node[i].Event = EVNT_SET_TIG_FBK_CALIB_POINT;
	node[i].var.Type = T_STRING;
	node[i].var.Var1ID = (h++);
	strcpy(node[i++].var.Format, "%s");

	node[i].pHeadNode	= (UDINT)&node[P_MODE_TIG_FBK_CALIB];
	node[i].Type = N_SCROLL;
	strcpy(node[i++].var.Format, " ******** ");

	node[i].pHeadNode	= (UDINT)&node[P_MODE_TIG_FBK_CALIB];
	node[i].Type = N_SCROLL;
	strcpy(node[i++].var.Format, " ******** ");

	node[i].pHeadNode	= (UDINT)&node[P_MODE_TIG_FBK_CALIB];
	node[i].Type = N_SCROLL +  N_EVENT ;
	node[i].Event = EVNT_LOAD_DEFAULT_CALIB;
	strcpy(node[i++].var.Format, "Load Default Calibr. !!!");

	// P_MODE_INDX_CALIB
	i= P_MODE_INDX_CALIB;			h=varSTRING_HMI_0;
	SetPageDict(&cfg->PagesDict[n++] , P_MODE_INDX_CALIB , "P_MODE_INDX_CALIB");

	/*
	node[i].pHeadNode	= (UDINT)&node[P_MODE_TVL_CALIB];
	node[i].Type = N_JUMP;
	node[i].JumpLineID = 0;
	node[i].pJumpNode = (UDINT)&node[P_MODE_CALIB];
	strcpy(node[i++].var.Format, "Cancel/Return ");
	*/

	node[i].pHeadNode	= (UDINT)&node[P_MODE_INDX_CALIB];
	node[i].Type = N_SCROLL;
	strcpy(node[i++].var.Format, "JOG BOTH");

	node[i].pHeadNode	= (UDINT)&node[P_MODE_INDX_CALIB];
	node[i].Type = N_SCROLL;
	strcpy(node[i++].var.Format, "JOG A");

	node[i].pHeadNode	= (UDINT)&node[P_MODE_INDX_CALIB];
	node[i].Type = N_SCROLL;
	strcpy(node[i++].var.Format, "JOG B");

	node[i].pHeadNode	= (UDINT)&node[P_MODE_INDX_CALIB];
	node[i].Type = N_SCROLL +  N_EVENT ;
	node[i].Event = EVNT_SET_INDX_ZERO;
	strcpy(node[i++].var.Format, "Set Zero");

	// P_MODE_TVL_CALIB_PAR
	i= P_MODE_TVL_CALIB_PAR;			h=varSTRING_HMI_0;
	SetPageDict(&cfg->PagesDict[n++] , P_MODE_TVL_CALIB_PAR , "P_MODE_TVL_CALIB_PAR");

	node[i].pHeadNode	= (UDINT)&node[P_MODE_TVL_CALIB_PAR];
	node[i].Type = N_SCROLL + N_EVENT;
	node[i].Event = EVNT_OK;
	node[i].var.Type = T_STRING;
	node[i].var.Var1ID = (h++);
	strcpy(node[i++].var.Format, "%s");

	node[i].pHeadNode	= (UDINT)&node[P_MODE_TVL_CALIB_PAR];
	node[i].Type = N_EDIT;
	node[i].var.Type = T_SCALED;
	node[i].var.Var1ID = parTVL_CalibVel1;
	//strcpy(node[i++].var.Format, "Low Vel: %s");
	strcpy(node[i++].var.Format, "%name%: %s");

	node[i].pHeadNode	= (UDINT)&node[P_MODE_TVL_CALIB_PAR];
	node[i].Type = N_EDIT;
	node[i].var.Type = T_SCALED;
	node[i].var.Var1ID = parTVL_CalibVel2;
	//strcpy(node[i++].var.Format, "High Vel: %s");
	strcpy(node[i++].var.Format, "%name%: %s");

	node[i].pHeadNode	= (UDINT)&node[P_MODE_TVL_CALIB_PAR];
	node[i].Type = N_EDIT;
	node[i].var.Type = T_SCALED;
	node[i].var.Var1ID = parGEN_CalibDist;
	//strcpy(node[i++].var.Format, "Dist.: %s");
	strcpy(node[i++].var.Format, "%name%: %s");

	node[i].pHeadNode	= (UDINT)&node[P_MODE_TVL_CALIB_PAR];
	node[i].Type = N_EDIT;
	node[i].var.Type = T_SCALED;
	node[i].var.Var1ID = parGEN_CalibDist_2;
	//strcpy(node[i++].var.Format, "Dist.: %s");
	strcpy(node[i++].var.Format, "%name%: %s");

	node[i].pHeadNode	= (UDINT)&node[P_MODE_TVL_CALIB_PAR];
	node[i].Type = N_SCROLL;
	node[i].var.Type = T_STRING;
	node[i].var.Var1ID = (h++);
	strcpy(node[i++].var.Format, "%s");

	node[i].pHeadNode	= (UDINT)&node[P_MODE_TVL_CALIB_PAR];
	node[i].Type = N_SCROLL + N_EVENT;
	node[i].Event = EVNT_CANCEL;
	node[i].var.Type = T_STRING;
	node[i].var.Var1ID = (h++);
	strcpy(node[i++].var.Format, "%s");

	// P_MODE_TVL_CALIB
	i= P_MODE_TVL_CALIB;			h=varSTRING_HMI_0;
	SetPageDict(&cfg->PagesDict[n++] , P_MODE_TVL_CALIB , "P_MODE_TVL_CALIB");

	/*
	node[i].pHeadNode	= (UDINT)&node[P_MODE_TVL_CALIB];
	node[i].Type = N_JUMP;
	node[i].JumpLineID = 0;
	node[i].pJumpNode = (UDINT)&node[P_MODE_TVL_CALIB_PAR];
	strcpy(node[i++].var.Format, "Cancel/Return ");
	*/

	node[i].pHeadNode	= (UDINT)&node[P_MODE_TVL_CALIB];
	node[i].Type = N_SCROLL +  N_EVENT ;
	node[i].Event = EVNT_CANCEL;
	node[i].var.Type = T_STRING;
	node[i].var.Var1ID = (h++);
	strcpy(node[i++].var.Format, "%s");

	node[i].pHeadNode	= (UDINT)&node[P_MODE_TVL_CALIB];
	node[i].Type = N_EDIT;
	node[i].var.Type = T_SCALED;
	node[i].var.Var1ID = parGEN_CalibTime1;
	//strcpy(node[i++].var.Format, "(1)Time Low Vel. FWD:   %s");
	strcpy(node[i++].var.Format, "%name%: %s");

	node[i].pHeadNode	= (UDINT)&node[P_MODE_TVL_CALIB];
	node[i].Type = N_EDIT;
	node[i].var.Type = T_SCALED;
	node[i].var.Var1ID = parGEN_CalibTime2;
	//strcpy(node[i++].var.Format, "(2)Time Low Vel. REV:   %s");
	strcpy(node[i++].var.Format, "%name%: %s");

	node[i].pHeadNode	= (UDINT)&node[P_MODE_TVL_CALIB];
	node[i].Type = N_EDIT;
	node[i].var.Type = T_SCALED;
	node[i].var.Var1ID = parGEN_CalibTime3;
	//strcpy(node[i++].var.Format, "(3)Time High Vel. FWD:   %s");
	strcpy(node[i++].var.Format, "%name%: %s");
```
